// TIA Portal V16 export
// export: Created 2021-11-12T13:32:42.386026Z, ExportSetting WithDefaults, DisplayName Totally Integrated Automation Portal, DisplayVersion V16 Update 3, DisplayName TIA Portal Version Control Interface, DisplayVersion V16 Update 2, DisplayName TIA Portal Openness, DisplayVersion V16 Update 3, DisplayName SINAMICS Startdrive Advanced, DisplayVersion V16 Update 5, DisplayName SINAMICS Startdrive G130, G150, S120, S150, SINAMICS MV, S210, DisplayVersion V16 Update 5, DisplayName SINAMICS Startdrive G110M, G120, G120C, G120D, G120P, G115D, DisplayVersion V16 Update 5, DisplayName STEP 7 Professional, DisplayVersion V16 Update 3, DisplayName STEP 7 Safety, DisplayVersion V16, DisplayName WinCC UA Professional, DisplayVersion V16 Update 3
FUNCTION_BLOCK "StationSCH1"   // FB25, LAD
{ S7_Optimized_Access := 'TRUE' }
VERSION : 0.1
// stored: AutoNumber true, IsIECCheckEnabled false, IsRetainMemResEnabled false, MemoryReserve 100, SetENOAutomatically false, UDAEnableTagReadback false
   VAR_INPUT
      IS_Inputs : "UDT_COMM_SCH1_CRS";
   END_VAR
   VAR_OUTPUT
      OS_Outputs : "UDT_COMM_CRS_SCH1";
      OS_Status : "UDT_SCH_Status_specific";
   END_VAR
   VAR_IN_OUT
      XS_Parameter : "UDT_SCH_Parameter";
      XS_HMICommand : "UDT_SCH_Command";
   END_VAR
   VAR
      SF_Alarm1 : "STD_DI_Mon";
      SF_Alarm2 : "STD_DI_Mon";
      SF_Alarm3 : "STD_DI_Mon";
      SF_Alarm4 : "STD_DI_Mon";
      SF_Alarm5 : "STD_DI_Mon";
      SF_Alarm6 : "STD_DI_Mon";
      SF_Alarm7 : "STD_DI_Mon";
      SF_Alarm8 : "STD_DI_Mon";
      SF_Alarm9 : "STD_DI_Mon";
      SF_QW180 { S7_SetPoint := 'True'} : "STD_CH_AO";
      SF_QW182 { S7_SetPoint := 'True'} : "STD_CH_AO";
      SF_QW184 { S7_SetPoint := 'True'} : "STD_CH_AO";
      SF_QW186 { S7_SetPoint := 'True'} : "STD_CH_AO";
      Edge { S7_SetPoint := 'True'} : Array[0..31] of Bool;   // Edge evalution
      ST_Die3Rdy : TON_TIME;
      ST_Die456Rdy : TON_TIME;
      ST_StartPulse { S7_SetPoint := 'True'} : TP_TIME;
   END_VAR
   VAR RETAIN
      SDI_PartID : DInt;
      SI_PartType : Int;
   END_VAR
   VAR
      SF_Alarm10 { S7_SetPoint := 'True'} : "STD_DI_Mon";
   END_VAR
   VAR_TEMP
      TB1PwrOk : Bool;
      TB1_ReqOnePart : Bool;   // Request to eject one part
      TB1_ReqAllParts : Bool;   // Request to eject all parts in row
      TI_BufferFreePos : Int;   // Number of free position in buffer
      TI_Index1 : Int;   // Index
      TI_Index2 : Int;   // Index
      TS_Parameter : "UDT_SCH_Parameter";
      TS_HMICommand : "UDT_SCH_Command";
      TR_TempUpperLim : Real;   // Upper limit of tool temperature
      TR_TempLowerLim : Real;   // Lower limit of tool temperature
      TDI_BrakeTestTime : DInt;   // Remaining time to brake test - Press [min]
   END_VAR
   VAR CONSTANT
      CT_DieRdy : Time := T#5m;
      CT_StartPulse : Time := T#1s;
      CR_BrakeTestWrn : Real := 10.0;   // [min]
   END_VAR
   VAR_TEMP   // added for the SCL form of the ladder/FBD networks
      _w1 : Bool;
      _w2 : Bool;
      _w3 : Bool;
      _w4 : Bool;
      _w5 : Bool;
      _w6 : Bool;
      _w7 : Bool;
      _w8 : Bool;
      _w9 : Bool;
      _w10 : Bool;
      _w11 : Bool;
      _w12 : Bool;
      _w13 : Bool;
      _w14 : Bool;
      _w15 : Bool;
   END_VAR
BEGIN

REGION Network 1: Clear temporary variables
END_REGION

REGION Network 2: Copy In/Out variables to temporary variables
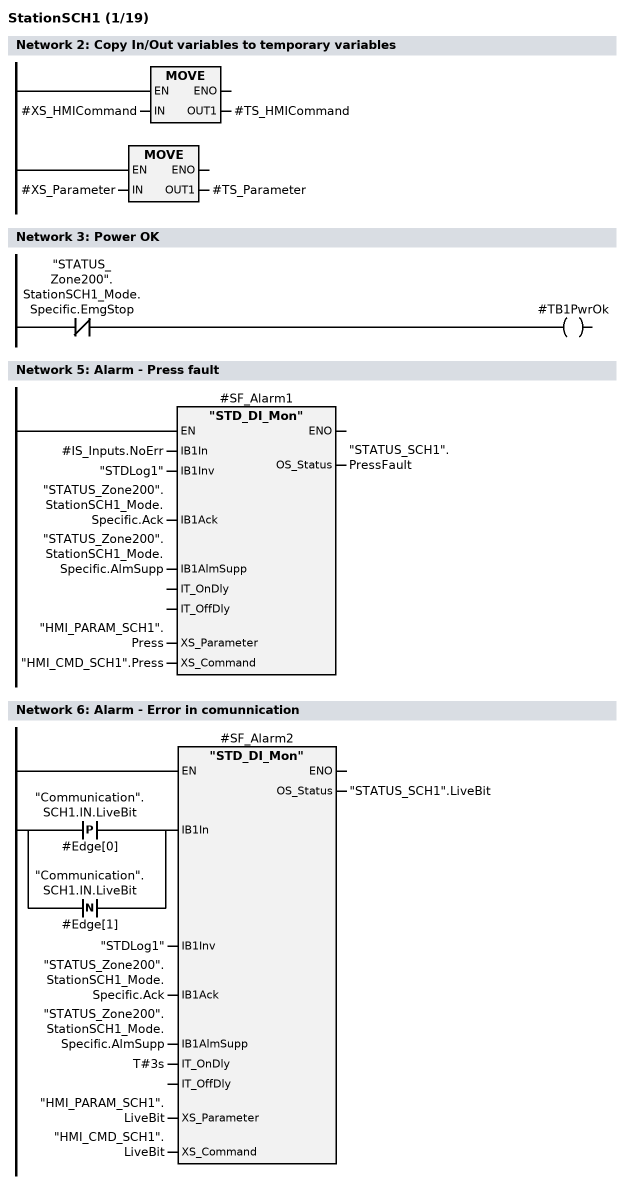
   RUNG wire#powerrail
      Move(in := #XS_HMICommand, out1 => #TS_HMICommand)
   END_RUNG
   RUNG wire#powerrail
      Move(in := #XS_Parameter, out1 => #TS_Parameter)
   END_RUNG
   // the same network as SCL:
   #TS_HMICommand := #XS_HMICommand;
   #TS_Parameter := #XS_Parameter;
END_REGION

REGION Network 3: Power OK
   RUNG wire#powerrail
      I_Contact( "STATUS_Zone200".StationSCH1_Mode.Specific.EmgStop )
      Coil( #TB1PwrOk )
   END_RUNG
   // the same network as SCL:
   #TB1PwrOk := NOT "STATUS_Zone200".StationSCH1_Mode.Specific.EmgStop;
END_REGION

REGION Network 4: *************** Alarms ***************
END_REGION

REGION Network 5: Alarm - Press fault
   RUNG wire#powerrail
      #SF_Alarm1(IB1In := #IS_Inputs.NoErr, IB1Inv := "STDLog1", IB1Ack := "STATUS_Zone200".StationSCH1_Mode.Specific.Ack, IB1AlmSupp := "STATUS_Zone200".StationSCH1_Mode.Specific.AlmSupp, IT_OnDly :=, IT_OffDly :=, XS_Parameter := "HMI_PARAM_SCH1".Press, XS_Command := "HMI_CMD_SCH1".Press, OS_Status => "STATUS_SCH1".PressFault)
   END_RUNG
   // the same network as SCL:
   #SF_Alarm1(IB1In := #IS_Inputs.NoErr,   // "STD_DI_Mon"
              IB1Inv := "STDLog1",
              IB1Ack := "STATUS_Zone200".StationSCH1_Mode.Specific.Ack,
              IB1AlmSupp := "STATUS_Zone200".StationSCH1_Mode.Specific.AlmSupp,
              XS_Parameter := "HMI_PARAM_SCH1".Press,
              XS_Command := "HMI_CMD_SCH1".Press,
              OS_Status => "STATUS_SCH1".PressFault);
END_REGION

REGION Network 6: Alarm - Error in comunnication
   RUNG wire#powerrail
      #SF_Alarm2(IB1In := wire#w1, IB1Inv := "STDLog1", IB1Ack := "STATUS_Zone200".StationSCH1_Mode.Specific.Ack, IB1AlmSupp := "STATUS_Zone200".StationSCH1_Mode.Specific.AlmSupp, IT_OnDly := T#3s, IT_OffDly :=, XS_Parameter := "HMI_PARAM_SCH1".LiveBit, XS_Command := "HMI_CMD_SCH1".LiveBit, OS_Status => "STATUS_SCH1".LiveBit)
   END_RUNG
   RUNG wire#powerrail
      P_Contact(operand := "Communication".SCH1.IN.LiveBit, bit := #Edge[0])
   END_RUNG wire#w1
   RUNG wire#powerrail
      N_Contact(operand := "Communication".SCH1.IN.LiveBit, bit := #Edge[1])
   END_RUNG wire#w1
   // the same network as SCL:
   #_w1 := "Communication".SCH1.IN.LiveBit AND NOT #Edge[0];   // rising edge of "Communication".SCH1.IN.LiveBit
   #Edge[0] := "Communication".SCH1.IN.LiveBit;
   #_w2 := NOT "Communication".SCH1.IN.LiveBit AND #Edge[1];   // falling edge of "Communication".SCH1.IN.LiveBit
   #Edge[1] := "Communication".SCH1.IN.LiveBit;
   #SF_Alarm2(IB1In := #_w1 OR #_w2,   // "STD_DI_Mon"
              IB1Inv := "STDLog1",
              IB1Ack := "STATUS_Zone200".StationSCH1_Mode.Specific.Ack,
              IB1AlmSupp := "STATUS_Zone200".StationSCH1_Mode.Specific.AlmSupp,
              IT_OnDly := T#3s,
              XS_Parameter := "HMI_PARAM_SCH1".LiveBit,
              XS_Command := "HMI_CMD_SCH1".LiveBit,
              OS_Status => "STATUS_SCH1".LiveBit);
END_REGION

REGION Network 7: Alarm - Tool heating 1 up - temperature is out of tolerance
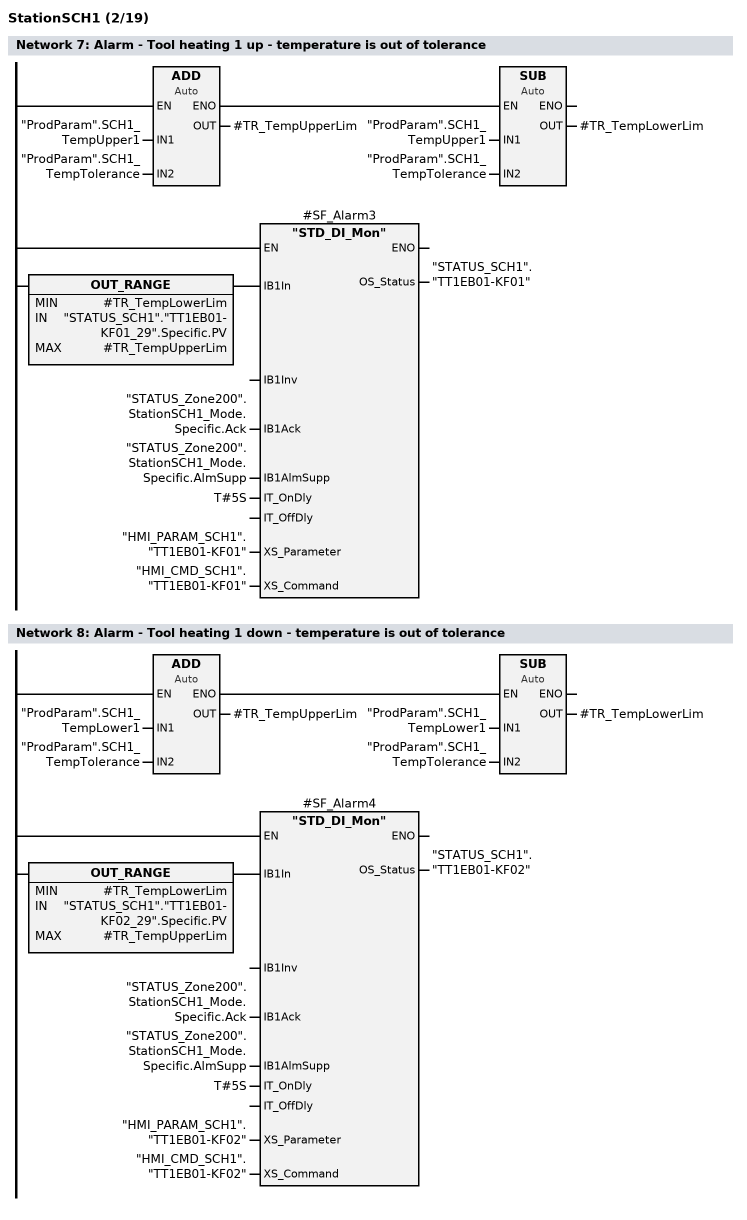
   #TR_TempUpperLim := "ProdParam".SCH1_TempUpper1 + "ProdParam".SCH1_TempTolerance;
   #TR_TempLowerLim := "ProdParam".SCH1_TempUpper1 - "ProdParam".SCH1_TempTolerance;
   #SF_Alarm3(IB1In := ("STATUS_SCH1"."TT1EB01-KF01_29".Specific.PV < #TR_TempLowerLim) OR ("STATUS_SCH1"."TT1EB01-KF01_29".Specific.PV > #TR_TempUpperLim),   // "STD_DI_Mon"
              IB1Ack := "STATUS_Zone200".StationSCH1_Mode.Specific.Ack,
              IB1AlmSupp := "STATUS_Zone200".StationSCH1_Mode.Specific.AlmSupp,
              IT_OnDly := T#5S,
              XS_Parameter := "HMI_PARAM_SCH1"."TT1EB01-KF01",
              XS_Command := "HMI_CMD_SCH1"."TT1EB01-KF01",
              OS_Status => "STATUS_SCH1"."TT1EB01-KF01");
END_REGION

REGION Network 8: Alarm - Tool heating 1 down - temperature is out of tolerance
   #TR_TempUpperLim := "ProdParam".SCH1_TempLower1 + "ProdParam".SCH1_TempTolerance;
   #TR_TempLowerLim := "ProdParam".SCH1_TempLower1 - "ProdParam".SCH1_TempTolerance;
   #SF_Alarm4(IB1In := ("STATUS_SCH1"."TT1EB01-KF02_29".Specific.PV < #TR_TempLowerLim) OR ("STATUS_SCH1"."TT1EB01-KF02_29".Specific.PV > #TR_TempUpperLim),   // "STD_DI_Mon"
              IB1Ack := "STATUS_Zone200".StationSCH1_Mode.Specific.Ack,
              IB1AlmSupp := "STATUS_Zone200".StationSCH1_Mode.Specific.AlmSupp,
              IT_OnDly := T#5S,
              XS_Parameter := "HMI_PARAM_SCH1"."TT1EB01-KF02",
              XS_Command := "HMI_CMD_SCH1"."TT1EB01-KF02",
              OS_Status => "STATUS_SCH1"."TT1EB01-KF02");
END_REGION

REGION Network 9: Alarm - Tool heating 2 up - temperature is out of tolerance
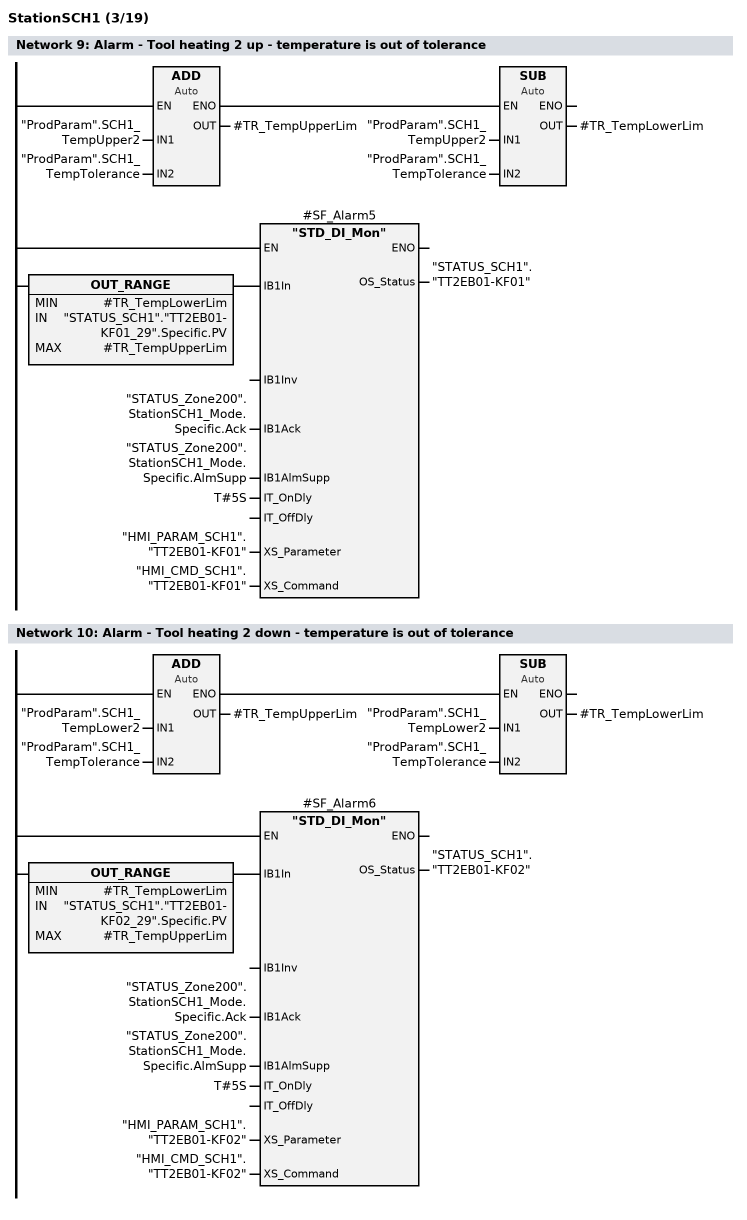
   #TR_TempUpperLim := "ProdParam".SCH1_TempUpper2 + "ProdParam".SCH1_TempTolerance;
   #TR_TempLowerLim := "ProdParam".SCH1_TempUpper2 - "ProdParam".SCH1_TempTolerance;
   #SF_Alarm5(IB1In := ("STATUS_SCH1"."TT2EB01-KF01_29".Specific.PV < #TR_TempLowerLim) OR ("STATUS_SCH1"."TT2EB01-KF01_29".Specific.PV > #TR_TempUpperLim),   // "STD_DI_Mon"
              IB1Ack := "STATUS_Zone200".StationSCH1_Mode.Specific.Ack,
              IB1AlmSupp := "STATUS_Zone200".StationSCH1_Mode.Specific.AlmSupp,
              IT_OnDly := T#5S,
              XS_Parameter := "HMI_PARAM_SCH1"."TT2EB01-KF01",
              XS_Command := "HMI_CMD_SCH1"."TT2EB01-KF01",
              OS_Status => "STATUS_SCH1"."TT2EB01-KF01");
END_REGION

REGION Network 10: Alarm - Tool heating 2 down - temperature is out of tolerance
   #TR_TempUpperLim := "ProdParam".SCH1_TempLower2 + "ProdParam".SCH1_TempTolerance;
   #TR_TempLowerLim := "ProdParam".SCH1_TempLower2 - "ProdParam".SCH1_TempTolerance;
   #SF_Alarm6(IB1In := ("STATUS_SCH1"."TT2EB01-KF02_29".Specific.PV < #TR_TempLowerLim) OR ("STATUS_SCH1"."TT2EB01-KF02_29".Specific.PV > #TR_TempUpperLim),   // "STD_DI_Mon"
              IB1Ack := "STATUS_Zone200".StationSCH1_Mode.Specific.Ack,
              IB1AlmSupp := "STATUS_Zone200".StationSCH1_Mode.Specific.AlmSupp,
              IT_OnDly := T#5S,
              XS_Parameter := "HMI_PARAM_SCH1"."TT2EB01-KF02",
              XS_Command := "HMI_CMD_SCH1"."TT2EB01-KF02",
              OS_Status => "STATUS_SCH1"."TT2EB01-KF02");
END_REGION

REGION Network 11: Alarm - Tool heating 1 - pump not running
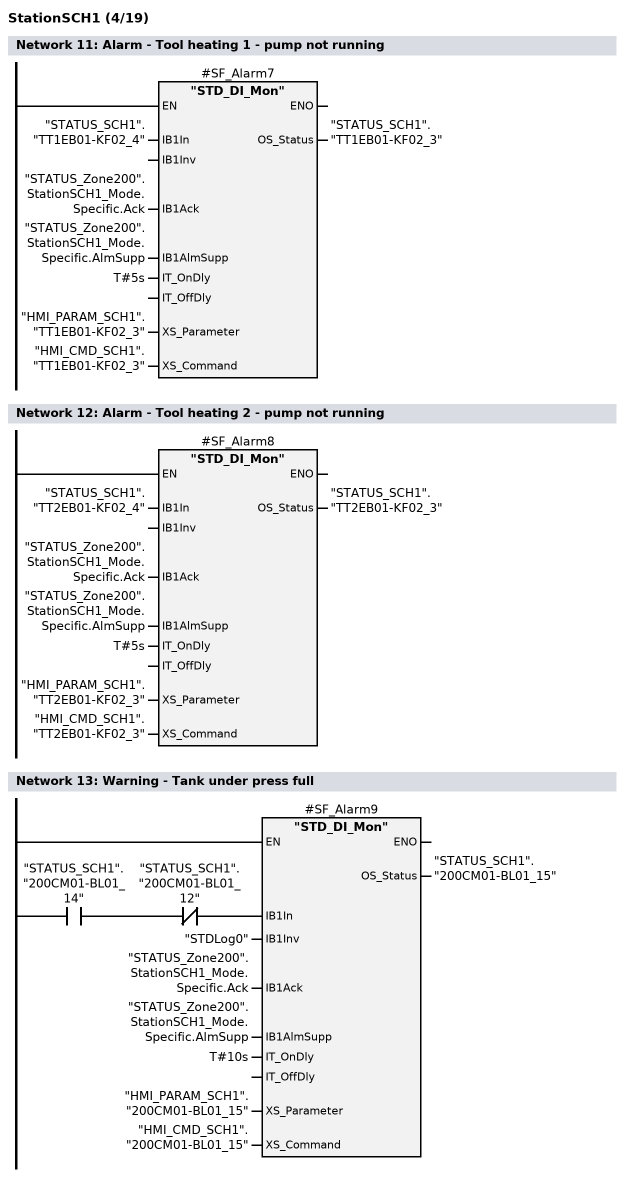
   RUNG wire#powerrail
      #SF_Alarm7(IB1In := "STATUS_SCH1"."TT1EB01-KF02_4", IB1Inv :=, IB1Ack := "STATUS_Zone200".StationSCH1_Mode.Specific.Ack, IB1AlmSupp := "STATUS_Zone200".StationSCH1_Mode.Specific.AlmSupp, IT_OnDly := T#5s, IT_OffDly :=, XS_Parameter := "HMI_PARAM_SCH1"."TT1EB01-KF02_3", XS_Command := "HMI_CMD_SCH1"."TT1EB01-KF02_3", OS_Status => "STATUS_SCH1"."TT1EB01-KF02_3")
   END_RUNG
   // the same network as SCL:
   #SF_Alarm7(IB1In := "STATUS_SCH1"."TT1EB01-KF02_4",   // "STD_DI_Mon"
              IB1Ack := "STATUS_Zone200".StationSCH1_Mode.Specific.Ack,
              IB1AlmSupp := "STATUS_Zone200".StationSCH1_Mode.Specific.AlmSupp,
              IT_OnDly := T#5s,
              XS_Parameter := "HMI_PARAM_SCH1"."TT1EB01-KF02_3",
              XS_Command := "HMI_CMD_SCH1"."TT1EB01-KF02_3",
              OS_Status => "STATUS_SCH1"."TT1EB01-KF02_3");
END_REGION

REGION Network 12: Alarm - Tool heating 2 - pump not running
   RUNG wire#powerrail
      #SF_Alarm8(IB1In := "STATUS_SCH1"."TT2EB01-KF02_4", IB1Inv :=, IB1Ack := "STATUS_Zone200".StationSCH1_Mode.Specific.Ack, IB1AlmSupp := "STATUS_Zone200".StationSCH1_Mode.Specific.AlmSupp, IT_OnDly := T#5s, IT_OffDly :=, XS_Parameter := "HMI_PARAM_SCH1"."TT2EB01-KF02_3", XS_Command := "HMI_CMD_SCH1"."TT2EB01-KF02_3", OS_Status => "STATUS_SCH1"."TT2EB01-KF02_3")
   END_RUNG
   // the same network as SCL:
   #SF_Alarm8(IB1In := "STATUS_SCH1"."TT2EB01-KF02_4",   // "STD_DI_Mon"
              IB1Ack := "STATUS_Zone200".StationSCH1_Mode.Specific.Ack,
              IB1AlmSupp := "STATUS_Zone200".StationSCH1_Mode.Specific.AlmSupp,
              IT_OnDly := T#5s,
              XS_Parameter := "HMI_PARAM_SCH1"."TT2EB01-KF02_3",
              XS_Command := "HMI_CMD_SCH1"."TT2EB01-KF02_3",
              OS_Status => "STATUS_SCH1"."TT2EB01-KF02_3");
END_REGION

REGION Network 13: Warning - Tank under press full
   RUNG wire#powerrail
      #SF_Alarm9(IB1In := wire#w1, IB1Inv := "STDLog0", IB1Ack := "STATUS_Zone200".StationSCH1_Mode.Specific.Ack, IB1AlmSupp := "STATUS_Zone200".StationSCH1_Mode.Specific.AlmSupp, IT_OnDly := T#10s, IT_OffDly :=, XS_Parameter := "HMI_PARAM_SCH1"."200CM01-BL01_15", XS_Command := "HMI_CMD_SCH1"."200CM01-BL01_15", OS_Status => "STATUS_SCH1"."200CM01-BL01_15")
   END_RUNG
   RUNG wire#powerrail
      Contact( "STATUS_SCH1"."200CM01-BL01_14" )
      I_Contact( "STATUS_SCH1"."200CM01-BL01_12" )
   END_RUNG wire#w1
   // the same network as SCL:
   #SF_Alarm9(IB1In := "STATUS_SCH1"."200CM01-BL01_14" AND NOT "STATUS_SCH1"."200CM01-BL01_12",   // "STD_DI_Mon"
              IB1Inv := "STDLog0",
              IB1Ack := "STATUS_Zone200".StationSCH1_Mode.Specific.Ack,
              IB1AlmSupp := "STATUS_Zone200".StationSCH1_Mode.Specific.AlmSupp,
              IT_OnDly := T#10s,
              XS_Parameter := "HMI_PARAM_SCH1"."200CM01-BL01_15",
              XS_Command := "HMI_CMD_SCH1"."200CM01-BL01_15",
              OS_Status => "STATUS_SCH1"."200CM01-BL01_15");
END_REGION

REGION Network 14: Warning - Brake test required
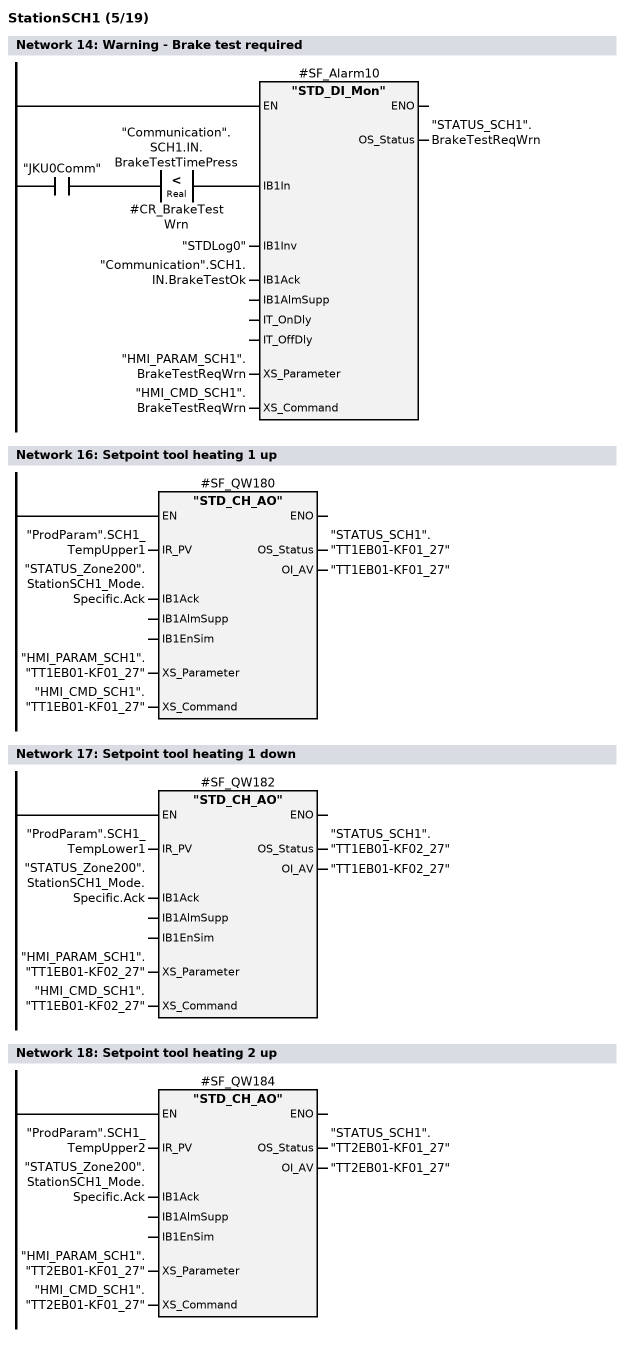
   RUNG wire#powerrail
      #SF_Alarm10(IB1In := wire#w1, IB1Inv := "STDLog0", IB1Ack := "Communication".SCH1.IN.BrakeTestOk, IB1AlmSupp :=, IT_OnDly :=, IT_OffDly :=, XS_Parameter := "HMI_PARAM_SCH1".BrakeTestReqWrn, XS_Command := "HMI_CMD_SCH1".BrakeTestReqWrn, OS_Status => "STATUS_SCH1".BrakeTestReqWrn)
   END_RUNG
   RUNG wire#powerrail
      Contact( "JKU0Comm" )
      { S7_Templates := "SrcType := Real" } LT_Contact(in1 := "Communication".SCH1.IN.BrakeTestTimePress, in2 := #CR_BrakeTestWrn)
   END_RUNG wire#w1
   // the same network as SCL:
   #SF_Alarm10(IB1In := "JKU0Comm" AND ("Communication".SCH1.IN.BrakeTestTimePress < #CR_BrakeTestWrn),   // "STD_DI_Mon"
               IB1Inv := "STDLog0",
               IB1Ack := "Communication".SCH1.IN.BrakeTestOk,
               XS_Parameter := "HMI_PARAM_SCH1".BrakeTestReqWrn,
               XS_Command := "HMI_CMD_SCH1".BrakeTestReqWrn,
               OS_Status => "STATUS_SCH1".BrakeTestReqWrn);
END_REGION

REGION Network 15: *************** Tool temperature setpoints ***************
END_REGION

REGION Network 16: Setpoint tool heating 1 up
   RUNG wire#powerrail
      #SF_QW180(IR_PV := "ProdParam".SCH1_TempUpper1, IB1Ack := "STATUS_Zone200".StationSCH1_Mode.Specific.Ack, IB1AlmSupp :=, IB1EnSim :=, XS_Parameter := "HMI_PARAM_SCH1"."TT1EB01-KF01_27", XS_Command := "HMI_CMD_SCH1"."TT1EB01-KF01_27", OS_Status => "STATUS_SCH1"."TT1EB01-KF01_27", OI_AV => "TT1EB01-KF01_27")
   END_RUNG
   // the same network as SCL:
   #SF_QW180(IR_PV := "ProdParam".SCH1_TempUpper1,   // "STD_CH_AO"
             IB1Ack := "STATUS_Zone200".StationSCH1_Mode.Specific.Ack,
             XS_Parameter := "HMI_PARAM_SCH1"."TT1EB01-KF01_27",
             XS_Command := "HMI_CMD_SCH1"."TT1EB01-KF01_27",
             OS_Status => "STATUS_SCH1"."TT1EB01-KF01_27",
             OI_AV => "TT1EB01-KF01_27");
END_REGION

REGION Network 17: Setpoint tool heating 1 down
   RUNG wire#powerrail
      #SF_QW182(IR_PV := "ProdParam".SCH1_TempLower1, IB1Ack := "STATUS_Zone200".StationSCH1_Mode.Specific.Ack, IB1AlmSupp :=, IB1EnSim :=, XS_Parameter := "HMI_PARAM_SCH1"."TT1EB01-KF02_27", XS_Command := "HMI_CMD_SCH1"."TT1EB01-KF02_27", OS_Status => "STATUS_SCH1"."TT1EB01-KF02_27", OI_AV => "TT1EB01-KF02_27")
   END_RUNG
   // the same network as SCL:
   #SF_QW182(IR_PV := "ProdParam".SCH1_TempLower1,   // "STD_CH_AO"
             IB1Ack := "STATUS_Zone200".StationSCH1_Mode.Specific.Ack,
             XS_Parameter := "HMI_PARAM_SCH1"."TT1EB01-KF02_27",
             XS_Command := "HMI_CMD_SCH1"."TT1EB01-KF02_27",
             OS_Status => "STATUS_SCH1"."TT1EB01-KF02_27",
             OI_AV => "TT1EB01-KF02_27");
END_REGION

REGION Network 18: Setpoint tool heating 2 up
   RUNG wire#powerrail
      #SF_QW184(IR_PV := "ProdParam".SCH1_TempUpper2, IB1Ack := "STATUS_Zone200".StationSCH1_Mode.Specific.Ack, IB1AlmSupp :=, IB1EnSim :=, XS_Parameter := "HMI_PARAM_SCH1"."TT2EB01-KF01_27", XS_Command := "HMI_CMD_SCH1"."TT2EB01-KF01_27", OS_Status => "STATUS_SCH1"."TT2EB01-KF01_27", OI_AV => "TT2EB01-KF01_27")
   END_RUNG
   // the same network as SCL:
   #SF_QW184(IR_PV := "ProdParam".SCH1_TempUpper2,   // "STD_CH_AO"
             IB1Ack := "STATUS_Zone200".StationSCH1_Mode.Specific.Ack,
             XS_Parameter := "HMI_PARAM_SCH1"."TT2EB01-KF01_27",
             XS_Command := "HMI_CMD_SCH1"."TT2EB01-KF01_27",
             OS_Status => "STATUS_SCH1"."TT2EB01-KF01_27",
             OI_AV => "TT2EB01-KF01_27");
END_REGION

REGION Network 19: Setpoint tool heating 2 down
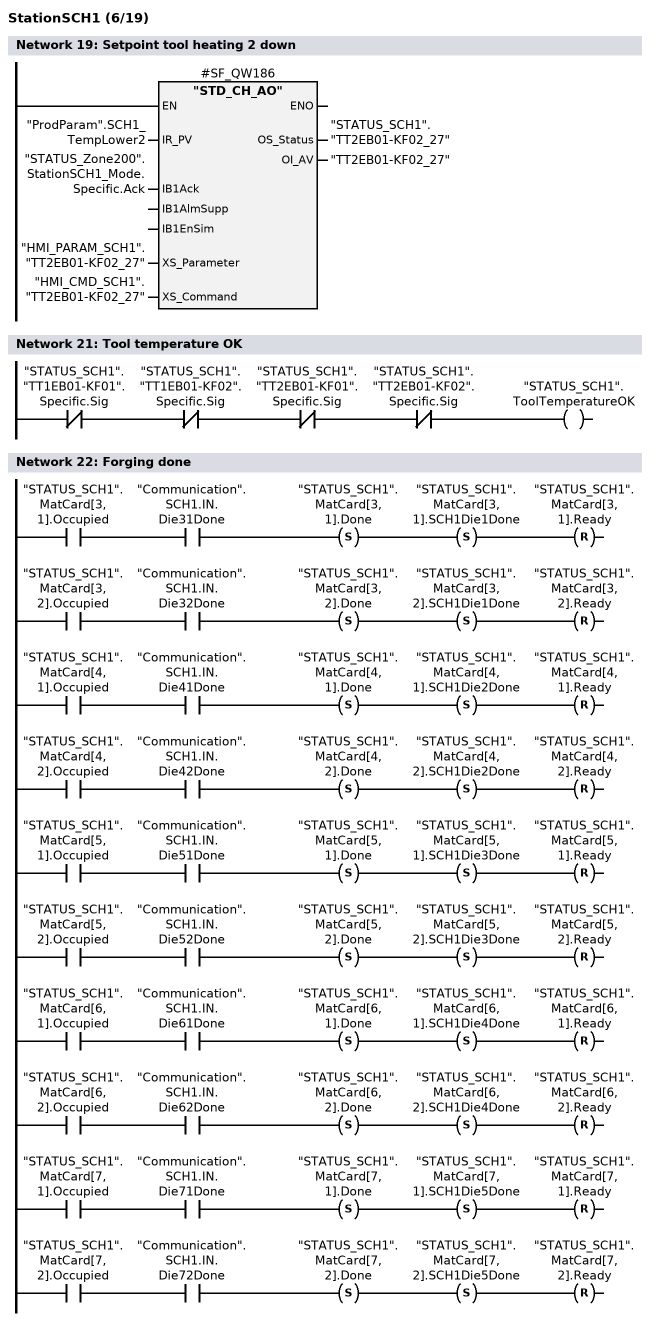
   RUNG wire#powerrail
      #SF_QW186(IR_PV := "ProdParam".SCH1_TempLower2, IB1Ack := "STATUS_Zone200".StationSCH1_Mode.Specific.Ack, IB1AlmSupp :=, IB1EnSim :=, XS_Parameter := "HMI_PARAM_SCH1"."TT2EB01-KF02_27", XS_Command := "HMI_CMD_SCH1"."TT2EB01-KF02_27", OS_Status => "STATUS_SCH1"."TT2EB01-KF02_27", OI_AV => "TT2EB01-KF02_27")
   END_RUNG
   // the same network as SCL:
   #SF_QW186(IR_PV := "ProdParam".SCH1_TempLower2,   // "STD_CH_AO"
             IB1Ack := "STATUS_Zone200".StationSCH1_Mode.Specific.Ack,
             XS_Parameter := "HMI_PARAM_SCH1"."TT2EB01-KF02_27",
             XS_Command := "HMI_CMD_SCH1"."TT2EB01-KF02_27",
             OS_Status => "STATUS_SCH1"."TT2EB01-KF02_27",
             OI_AV => "TT2EB01-KF02_27");
END_REGION

REGION Network 20: *************** States ***************
END_REGION

REGION Network 21: Tool temperature OK
   RUNG wire#powerrail
      I_Contact( "STATUS_SCH1"."TT1EB01-KF01".Specific.Sig )
      I_Contact( "STATUS_SCH1"."TT1EB01-KF02".Specific.Sig )
      I_Contact( "STATUS_SCH1"."TT2EB01-KF01".Specific.Sig )
      I_Contact( "STATUS_SCH1"."TT2EB01-KF02".Specific.Sig )
      Coil( "STATUS_SCH1".ToolTemperatureOK )
   END_RUNG
   // the same network as SCL:
   "STATUS_SCH1".ToolTemperatureOK := NOT "STATUS_SCH1"."TT1EB01-KF01".Specific.Sig AND NOT "STATUS_SCH1"."TT1EB01-KF02".Specific.Sig AND NOT "STATUS_SCH1"."TT2EB01-KF01".Specific.Sig AND NOT "STATUS_SCH1"."TT2EB01-KF02".Specific.Sig;
END_REGION

REGION Network 22: Forging done
   RUNG wire#powerrail
      Contact( "STATUS_SCH1".MatCard[3, 1].Occupied )
      Contact( "Communication".SCH1.IN.Die31Done )
      S_Coil( "STATUS_SCH1".MatCard[3, 1].Done )
      S_Coil( "STATUS_SCH1".MatCard[3, 1].SCH1Die1Done )
      R_Coil( "STATUS_SCH1".MatCard[3, 1].Ready )
   END_RUNG
   RUNG wire#powerrail
      Contact( "STATUS_SCH1".MatCard[3, 2].Occupied )
      Contact( "Communication".SCH1.IN.Die32Done )
      S_Coil( "STATUS_SCH1".MatCard[3, 2].Done )
      S_Coil( "STATUS_SCH1".MatCard[3, 2].SCH1Die1Done )
      R_Coil( "STATUS_SCH1".MatCard[3, 2].Ready )
   END_RUNG
   RUNG wire#powerrail
      Contact( "STATUS_SCH1".MatCard[4, 1].Occupied )
      Contact( "Communication".SCH1.IN.Die41Done )
      S_Coil( "STATUS_SCH1".MatCard[4, 1].Done )
      S_Coil( "STATUS_SCH1".MatCard[4, 1].SCH1Die2Done )
      R_Coil( "STATUS_SCH1".MatCard[4, 1].Ready )
   END_RUNG
   RUNG wire#powerrail
      Contact( "STATUS_SCH1".MatCard[4, 2].Occupied )
      Contact( "Communication".SCH1.IN.Die42Done )
      S_Coil( "STATUS_SCH1".MatCard[4, 2].Done )
      S_Coil( "STATUS_SCH1".MatCard[4, 2].SCH1Die2Done )
      R_Coil( "STATUS_SCH1".MatCard[4, 2].Ready )
   END_RUNG
   RUNG wire#powerrail
      Contact( "STATUS_SCH1".MatCard[5, 1].Occupied )
      Contact( "Communication".SCH1.IN.Die51Done )
      S_Coil( "STATUS_SCH1".MatCard[5, 1].Done )
      S_Coil( "STATUS_SCH1".MatCard[5, 1].SCH1Die3Done )
      R_Coil( "STATUS_SCH1".MatCard[5, 1].Ready )
   END_RUNG
   RUNG wire#powerrail
      Contact( "STATUS_SCH1".MatCard[5, 2].Occupied )
      Contact( "Communication".SCH1.IN.Die52Done )
      S_Coil( "STATUS_SCH1".MatCard[5, 2].Done )
      S_Coil( "STATUS_SCH1".MatCard[5, 2].SCH1Die3Done )
      R_Coil( "STATUS_SCH1".MatCard[5, 2].Ready )
   END_RUNG
   RUNG wire#powerrail
      Contact( "STATUS_SCH1".MatCard[6, 1].Occupied )
      Contact( "Communication".SCH1.IN.Die61Done )
      S_Coil( "STATUS_SCH1".MatCard[6, 1].Done )
      S_Coil( "STATUS_SCH1".MatCard[6, 1].SCH1Die4Done )
      R_Coil( "STATUS_SCH1".MatCard[6, 1].Ready )
   END_RUNG
   RUNG wire#powerrail
      Contact( "STATUS_SCH1".MatCard[6, 2].Occupied )
      Contact( "Communication".SCH1.IN.Die62Done )
      S_Coil( "STATUS_SCH1".MatCard[6, 2].Done )
      S_Coil( "STATUS_SCH1".MatCard[6, 2].SCH1Die4Done )
      R_Coil( "STATUS_SCH1".MatCard[6, 2].Ready )
   END_RUNG
   RUNG wire#powerrail
      Contact( "STATUS_SCH1".MatCard[7, 1].Occupied )
      Contact( "Communication".SCH1.IN.Die71Done )
      S_Coil( "STATUS_SCH1".MatCard[7, 1].Done )
      S_Coil( "STATUS_SCH1".MatCard[7, 1].SCH1Die5Done )
      R_Coil( "STATUS_SCH1".MatCard[7, 1].Ready )
   END_RUNG
   RUNG wire#powerrail
      Contact( "STATUS_SCH1".MatCard[7, 2].Occupied )
      Contact( "Communication".SCH1.IN.Die72Done )
      S_Coil( "STATUS_SCH1".MatCard[7, 2].Done )
      S_Coil( "STATUS_SCH1".MatCard[7, 2].SCH1Die5Done )
      R_Coil( "STATUS_SCH1".MatCard[7, 2].Ready )
   END_RUNG
   // the same network as SCL:
   #_w1 := "STATUS_SCH1".MatCard[3, 1].Occupied AND "Communication".SCH1.IN.Die31Done;
   IF #_w1 THEN
       "STATUS_SCH1".MatCard[3, 1].Done := TRUE;
       "STATUS_SCH1".MatCard[3, 1].SCH1Die1Done := TRUE;
       "STATUS_SCH1".MatCard[3, 1].Ready := FALSE;
   END_IF;
   #_w2 := "STATUS_SCH1".MatCard[3, 2].Occupied AND "Communication".SCH1.IN.Die32Done;
   IF #_w2 THEN
       "STATUS_SCH1".MatCard[3, 2].Done := TRUE;
       "STATUS_SCH1".MatCard[3, 2].SCH1Die1Done := TRUE;
       "STATUS_SCH1".MatCard[3, 2].Ready := FALSE;
   END_IF;
   #_w3 := "STATUS_SCH1".MatCard[4, 1].Occupied AND "Communication".SCH1.IN.Die41Done;
   IF #_w3 THEN
       "STATUS_SCH1".MatCard[4, 1].Done := TRUE;
       "STATUS_SCH1".MatCard[4, 1].SCH1Die2Done := TRUE;
       "STATUS_SCH1".MatCard[4, 1].Ready := FALSE;
   END_IF;
   #_w4 := "STATUS_SCH1".MatCard[4, 2].Occupied AND "Communication".SCH1.IN.Die42Done;
   IF #_w4 THEN
       "STATUS_SCH1".MatCard[4, 2].Done := TRUE;
       "STATUS_SCH1".MatCard[4, 2].SCH1Die2Done := TRUE;
       "STATUS_SCH1".MatCard[4, 2].Ready := FALSE;
   END_IF;
   #_w5 := "STATUS_SCH1".MatCard[5, 1].Occupied AND "Communication".SCH1.IN.Die51Done;
   IF #_w5 THEN
       "STATUS_SCH1".MatCard[5, 1].Done := TRUE;
       "STATUS_SCH1".MatCard[5, 1].SCH1Die3Done := TRUE;
       "STATUS_SCH1".MatCard[5, 1].Ready := FALSE;
   END_IF;
   #_w6 := "STATUS_SCH1".MatCard[5, 2].Occupied AND "Communication".SCH1.IN.Die52Done;
   IF #_w6 THEN
       "STATUS_SCH1".MatCard[5, 2].Done := TRUE;
       "STATUS_SCH1".MatCard[5, 2].SCH1Die3Done := TRUE;
       "STATUS_SCH1".MatCard[5, 2].Ready := FALSE;
   END_IF;
   #_w7 := "STATUS_SCH1".MatCard[6, 1].Occupied AND "Communication".SCH1.IN.Die61Done;
   IF #_w7 THEN
       "STATUS_SCH1".MatCard[6, 1].Done := TRUE;
       "STATUS_SCH1".MatCard[6, 1].SCH1Die4Done := TRUE;
       "STATUS_SCH1".MatCard[6, 1].Ready := FALSE;
   END_IF;
   #_w8 := "STATUS_SCH1".MatCard[6, 2].Occupied AND "Communication".SCH1.IN.Die62Done;
   IF #_w8 THEN
       "STATUS_SCH1".MatCard[6, 2].Done := TRUE;
       "STATUS_SCH1".MatCard[6, 2].SCH1Die4Done := TRUE;
       "STATUS_SCH1".MatCard[6, 2].Ready := FALSE;
   END_IF;
   #_w9 := "STATUS_SCH1".MatCard[7, 1].Occupied AND "Communication".SCH1.IN.Die71Done;
   IF #_w9 THEN
       "STATUS_SCH1".MatCard[7, 1].Done := TRUE;
       "STATUS_SCH1".MatCard[7, 1].SCH1Die5Done := TRUE;
       "STATUS_SCH1".MatCard[7, 1].Ready := FALSE;
   END_IF;
   #_w10 := "STATUS_SCH1".MatCard[7, 2].Occupied AND "Communication".SCH1.IN.Die72Done;
   IF #_w10 THEN
       "STATUS_SCH1".MatCard[7, 2].Done := TRUE;
       "STATUS_SCH1".MatCard[7, 2].SCH1Die5Done := TRUE;
       "STATUS_SCH1".MatCard[7, 2].Ready := FALSE;
   END_IF;
END_REGION

REGION Network 23 (SCL): Tech. time evaluation
   IF "STDEdge_1s" THEN
       FOR #TI_Index1 := 3 TO 7 DO
           FOR #TI_Index2 := 1 TO 2 DO
               IF "STATUS_SCH1".MatCard[#TI_Index1, #TI_Index2].Occupied THEN
                   "MTS_UpdateTimeInPress"(IB1Clock_1s := "STDEdge_1s",
                                           XS_Position := "STATUS_SCH1".MatCard[#TI_Index1, #TI_Index2]);
               END_IF;
           END_FOR;
       END_FOR;
   END_IF;
END_REGION

REGION Network 24: Output conveyor part counter
END_REGION

REGION Network 25: Brake test time
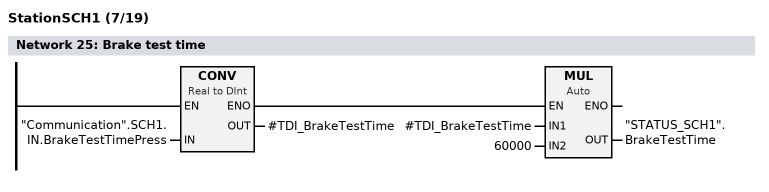
   RUNG wire#powerrail
      { S7_Templates := "[SrcType := Real, DestType := DInt]"; S7_GenerateENO := "TRUE" } Convert(in := "Communication".SCH1.IN.BrakeTestTimePress, out => #TDI_BrakeTestTime)
      { S7_GenerateENO := "TRUE" } Mul(in1 := #TDI_BrakeTestTime, in2 := 60000, out => "STATUS_SCH1".BrakeTestTime)
   END_RUNG
   // the same network as SCL:
   // ENO of a box is taken as its EN; it also drops when the box reports an error
   #TDI_BrakeTestTime := REAL_TO_DINT("Communication".SCH1.IN.BrakeTestTimePress);
   "STATUS_SCH1".BrakeTestTime := #TDI_BrakeTestTime * 60000;
END_REGION

REGION Network 26: *************** Material flow ***************
END_REGION

REGION Network 27: Clear positions and map - commands
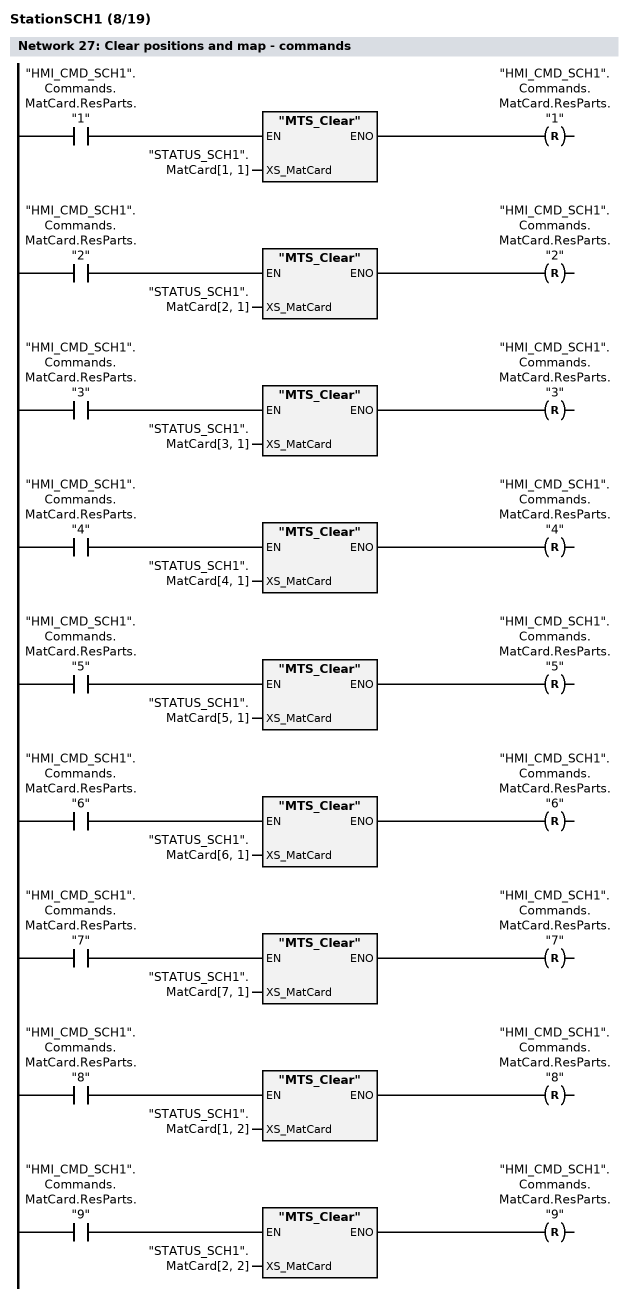
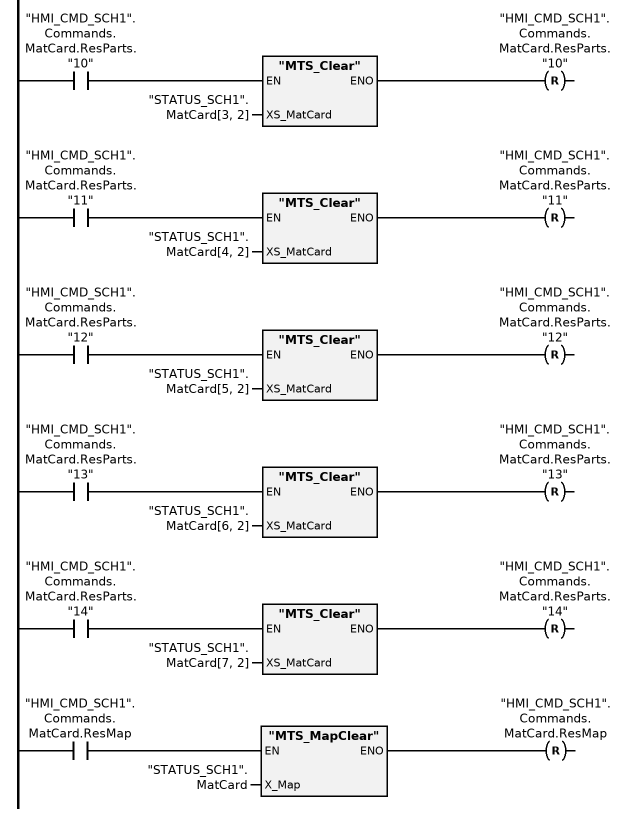
   RUNG wire#powerrail
      Contact( "HMI_CMD_SCH1".Commands.MatCard.ResParts."1" )
      "MTS_Clear"(XS_MatCard := "STATUS_SCH1".MatCard[1, 1])
      R_Coil( "HMI_CMD_SCH1".Commands.MatCard.ResParts."1" )
   END_RUNG
   RUNG wire#powerrail
      Contact( "HMI_CMD_SCH1".Commands.MatCard.ResParts."2" )
      "MTS_Clear"(XS_MatCard := "STATUS_SCH1".MatCard[2, 1])
      R_Coil( "HMI_CMD_SCH1".Commands.MatCard.ResParts."2" )
   END_RUNG
   RUNG wire#powerrail
      Contact( "HMI_CMD_SCH1".Commands.MatCard.ResParts."3" )
      "MTS_Clear"(XS_MatCard := "STATUS_SCH1".MatCard[3, 1])
      R_Coil( "HMI_CMD_SCH1".Commands.MatCard.ResParts."3" )
   END_RUNG
   RUNG wire#powerrail
      Contact( "HMI_CMD_SCH1".Commands.MatCard.ResParts."4" )
      "MTS_Clear"(XS_MatCard := "STATUS_SCH1".MatCard[4, 1])
      R_Coil( "HMI_CMD_SCH1".Commands.MatCard.ResParts."4" )
   END_RUNG
   RUNG wire#powerrail
      Contact( "HMI_CMD_SCH1".Commands.MatCard.ResParts."5" )
      "MTS_Clear"(XS_MatCard := "STATUS_SCH1".MatCard[5, 1])
      R_Coil( "HMI_CMD_SCH1".Commands.MatCard.ResParts."5" )
   END_RUNG
   RUNG wire#powerrail
      Contact( "HMI_CMD_SCH1".Commands.MatCard.ResParts."6" )
      "MTS_Clear"(XS_MatCard := "STATUS_SCH1".MatCard[6, 1])
      R_Coil( "HMI_CMD_SCH1".Commands.MatCard.ResParts."6" )
   END_RUNG
   RUNG wire#powerrail
      Contact( "HMI_CMD_SCH1".Commands.MatCard.ResParts."7" )
      "MTS_Clear"(XS_MatCard := "STATUS_SCH1".MatCard[7, 1])
      R_Coil( "HMI_CMD_SCH1".Commands.MatCard.ResParts."7" )
   END_RUNG
   RUNG wire#powerrail
      Contact( "HMI_CMD_SCH1".Commands.MatCard.ResParts."8" )
      "MTS_Clear"(XS_MatCard := "STATUS_SCH1".MatCard[1, 2])
      R_Coil( "HMI_CMD_SCH1".Commands.MatCard.ResParts."8" )
   END_RUNG
   RUNG wire#powerrail
      Contact( "HMI_CMD_SCH1".Commands.MatCard.ResParts."9" )
      "MTS_Clear"(XS_MatCard := "STATUS_SCH1".MatCard[2, 2])
      R_Coil( "HMI_CMD_SCH1".Commands.MatCard.ResParts."9" )
   END_RUNG
   RUNG wire#powerrail
      Contact( "HMI_CMD_SCH1".Commands.MatCard.ResParts."10" )
      "MTS_Clear"(XS_MatCard := "STATUS_SCH1".MatCard[3, 2])
      R_Coil( "HMI_CMD_SCH1".Commands.MatCard.ResParts."10" )
   END_RUNG
   RUNG wire#powerrail
      Contact( "HMI_CMD_SCH1".Commands.MatCard.ResParts."11" )
      "MTS_Clear"(XS_MatCard := "STATUS_SCH1".MatCard[4, 2])
      R_Coil( "HMI_CMD_SCH1".Commands.MatCard.ResParts."11" )
   END_RUNG
   RUNG wire#powerrail
      Contact( "HMI_CMD_SCH1".Commands.MatCard.ResParts."12" )
      "MTS_Clear"(XS_MatCard := "STATUS_SCH1".MatCard[5, 2])
      R_Coil( "HMI_CMD_SCH1".Commands.MatCard.ResParts."12" )
   END_RUNG
   RUNG wire#powerrail
      Contact( "HMI_CMD_SCH1".Commands.MatCard.ResParts."13" )
      "MTS_Clear"(XS_MatCard := "STATUS_SCH1".MatCard[6, 2])
      R_Coil( "HMI_CMD_SCH1".Commands.MatCard.ResParts."13" )
   END_RUNG
   RUNG wire#powerrail
      Contact( "HMI_CMD_SCH1".Commands.MatCard.ResParts."14" )
      "MTS_Clear"(XS_MatCard := "STATUS_SCH1".MatCard[7, 2])
      R_Coil( "HMI_CMD_SCH1".Commands.MatCard.ResParts."14" )
   END_RUNG
   RUNG wire#powerrail
      Contact( "HMI_CMD_SCH1".Commands.MatCard.ResMap )
      "MTS_MapClear"(X_Map := "STATUS_SCH1".MatCard)
      R_Coil( "HMI_CMD_SCH1".Commands.MatCard.ResMap )
   END_RUNG
   // the same network as SCL:
   "MTS_Clear"(EN := "HMI_CMD_SCH1".Commands.MatCard.ResParts."1",
               XS_MatCard := "STATUS_SCH1".MatCard[1, 1],
               ENO => #_w1);
   IF #_w1 THEN "HMI_CMD_SCH1".Commands.MatCard.ResParts."1" := FALSE; END_IF;
   "MTS_Clear"(EN := "HMI_CMD_SCH1".Commands.MatCard.ResParts."2",
               XS_MatCard := "STATUS_SCH1".MatCard[2, 1],
               ENO => #_w2);
   IF #_w2 THEN "HMI_CMD_SCH1".Commands.MatCard.ResParts."2" := FALSE; END_IF;
   "MTS_Clear"(EN := "HMI_CMD_SCH1".Commands.MatCard.ResParts."3",
               XS_MatCard := "STATUS_SCH1".MatCard[3, 1],
               ENO => #_w3);
   IF #_w3 THEN "HMI_CMD_SCH1".Commands.MatCard.ResParts."3" := FALSE; END_IF;
   "MTS_Clear"(EN := "HMI_CMD_SCH1".Commands.MatCard.ResParts."4",
               XS_MatCard := "STATUS_SCH1".MatCard[4, 1],
               ENO => #_w4);
   IF #_w4 THEN "HMI_CMD_SCH1".Commands.MatCard.ResParts."4" := FALSE; END_IF;
   "MTS_Clear"(EN := "HMI_CMD_SCH1".Commands.MatCard.ResParts."5",
               XS_MatCard := "STATUS_SCH1".MatCard[5, 1],
               ENO => #_w5);
   IF #_w5 THEN "HMI_CMD_SCH1".Commands.MatCard.ResParts."5" := FALSE; END_IF;
   "MTS_Clear"(EN := "HMI_CMD_SCH1".Commands.MatCard.ResParts."6",
               XS_MatCard := "STATUS_SCH1".MatCard[6, 1],
               ENO => #_w6);
   IF #_w6 THEN "HMI_CMD_SCH1".Commands.MatCard.ResParts."6" := FALSE; END_IF;
   "MTS_Clear"(EN := "HMI_CMD_SCH1".Commands.MatCard.ResParts."7",
               XS_MatCard := "STATUS_SCH1".MatCard[7, 1],
               ENO => #_w7);
   IF #_w7 THEN "HMI_CMD_SCH1".Commands.MatCard.ResParts."7" := FALSE; END_IF;
   "MTS_Clear"(EN := "HMI_CMD_SCH1".Commands.MatCard.ResParts."8",
               XS_MatCard := "STATUS_SCH1".MatCard[1, 2],
               ENO => #_w8);
   IF #_w8 THEN "HMI_CMD_SCH1".Commands.MatCard.ResParts."8" := FALSE; END_IF;
   "MTS_Clear"(EN := "HMI_CMD_SCH1".Commands.MatCard.ResParts."9",
               XS_MatCard := "STATUS_SCH1".MatCard[2, 2],
               ENO => #_w9);
   IF #_w9 THEN "HMI_CMD_SCH1".Commands.MatCard.ResParts."9" := FALSE; END_IF;
   "MTS_Clear"(EN := "HMI_CMD_SCH1".Commands.MatCard.ResParts."10",
               XS_MatCard := "STATUS_SCH1".MatCard[3, 2],
               ENO => #_w10);
   IF #_w10 THEN "HMI_CMD_SCH1".Commands.MatCard.ResParts."10" := FALSE; END_IF;
   "MTS_Clear"(EN := "HMI_CMD_SCH1".Commands.MatCard.ResParts."11",
               XS_MatCard := "STATUS_SCH1".MatCard[4, 2],
               ENO => #_w11);
   IF #_w11 THEN "HMI_CMD_SCH1".Commands.MatCard.ResParts."11" := FALSE; END_IF;
   "MTS_Clear"(EN := "HMI_CMD_SCH1".Commands.MatCard.ResParts."12",
               XS_MatCard := "STATUS_SCH1".MatCard[5, 2],
               ENO => #_w12);
   IF #_w12 THEN "HMI_CMD_SCH1".Commands.MatCard.ResParts."12" := FALSE; END_IF;
   "MTS_Clear"(EN := "HMI_CMD_SCH1".Commands.MatCard.ResParts."13",
               XS_MatCard := "STATUS_SCH1".MatCard[6, 2],
               ENO => #_w13);
   IF #_w13 THEN "HMI_CMD_SCH1".Commands.MatCard.ResParts."13" := FALSE; END_IF;
   "MTS_Clear"(EN := "HMI_CMD_SCH1".Commands.MatCard.ResParts."14",
               XS_MatCard := "STATUS_SCH1".MatCard[7, 2],
               ENO => #_w14);
   IF #_w14 THEN "HMI_CMD_SCH1".Commands.MatCard.ResParts."14" := FALSE; END_IF;
   "MTS_MapClear"(EN := "HMI_CMD_SCH1".Commands.MatCard.ResMap, X_Map := "STATUS_SCH1".MatCard, ENO => #_w15);
   IF #_w15 THEN "HMI_CMD_SCH1".Commands.MatCard.ResMap := FALSE; END_IF;
END_REGION

REGION Network 28: Set positions in press - init
   // "JSA0Comm" - change when recipes done
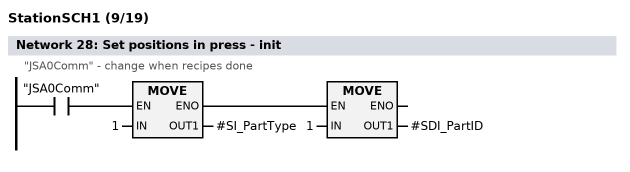
   RUNG wire#powerrail
      Contact( "JSA0Comm" )
      Move(in := 1, out1 => #SI_PartType)
      Move(in := 1, out1 => #SDI_PartID)
   END_RUNG
   // the same network as SCL:
   IF "JSA0Comm" THEN
       #SI_PartType := 1;
       #SDI_PartID := 1;
   END_IF;
END_REGION

REGION Network 29: Set positions in press - commands
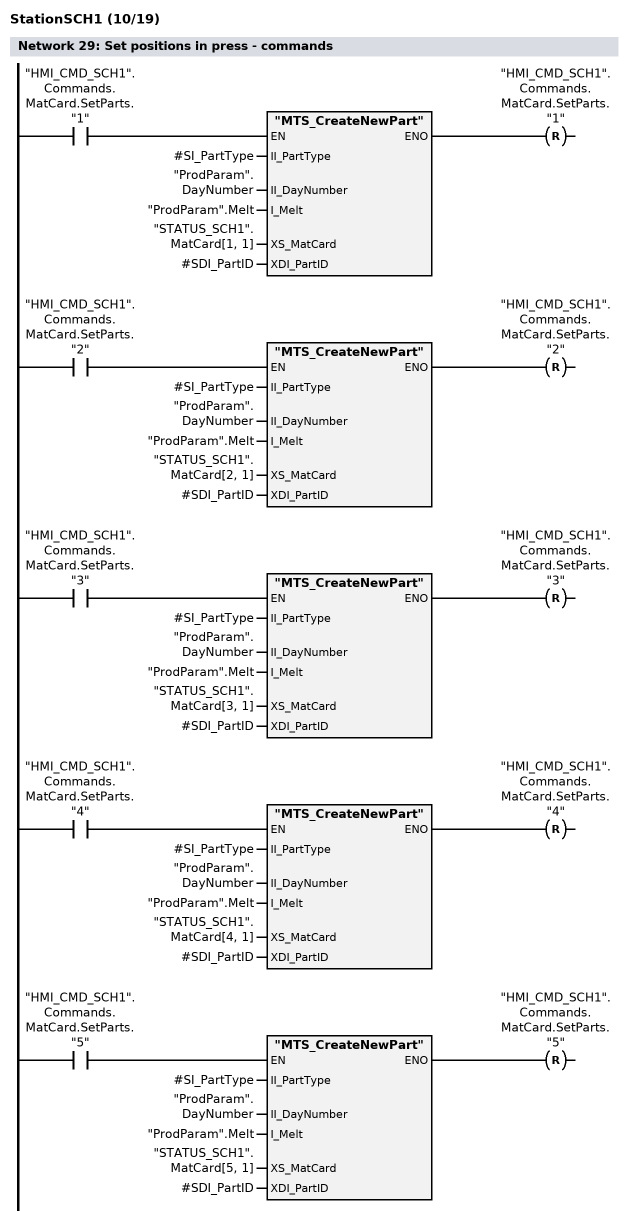
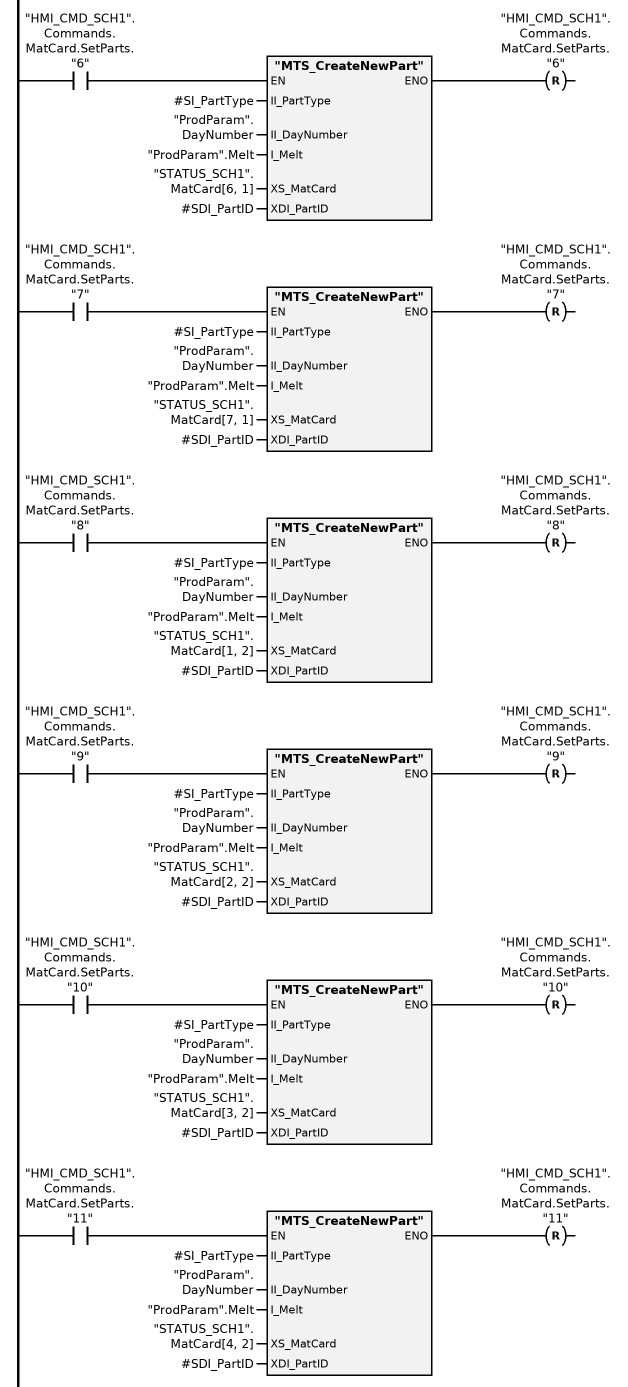
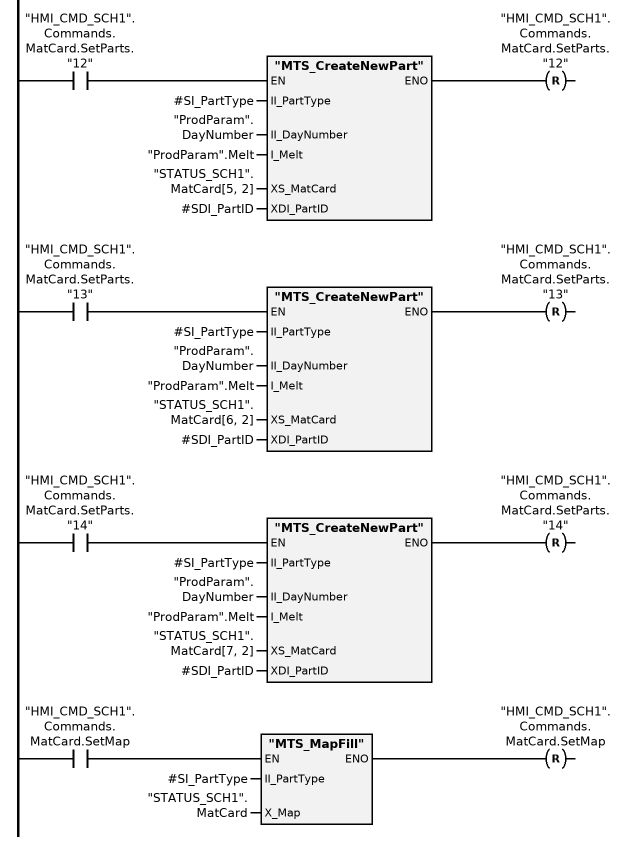
   RUNG wire#powerrail
      Contact( "HMI_CMD_SCH1".Commands.MatCard.SetParts."1" )
      "MTS_CreateNewPart"(II_PartType := #SI_PartType, II_DayNumber := "ProdParam".DayNumber, I_Melt := "ProdParam".Melt, XS_MatCard := "STATUS_SCH1".MatCard[1, 1], XDI_PartID := #SDI_PartID)
      R_Coil( "HMI_CMD_SCH1".Commands.MatCard.SetParts."1" )
   END_RUNG
   RUNG wire#powerrail
      Contact( "HMI_CMD_SCH1".Commands.MatCard.SetParts."2" )
      "MTS_CreateNewPart"(II_PartType := #SI_PartType, II_DayNumber := "ProdParam".DayNumber, I_Melt := "ProdParam".Melt, XS_MatCard := "STATUS_SCH1".MatCard[2, 1], XDI_PartID := #SDI_PartID)
      R_Coil( "HMI_CMD_SCH1".Commands.MatCard.SetParts."2" )
   END_RUNG
   RUNG wire#powerrail
      Contact( "HMI_CMD_SCH1".Commands.MatCard.SetParts."3" )
      "MTS_CreateNewPart"(II_PartType := #SI_PartType, II_DayNumber := "ProdParam".DayNumber, I_Melt := "ProdParam".Melt, XS_MatCard := "STATUS_SCH1".MatCard[3, 1], XDI_PartID := #SDI_PartID)
      R_Coil( "HMI_CMD_SCH1".Commands.MatCard.SetParts."3" )
   END_RUNG
   RUNG wire#powerrail
      Contact( "HMI_CMD_SCH1".Commands.MatCard.SetParts."4" )
      "MTS_CreateNewPart"(II_PartType := #SI_PartType, II_DayNumber := "ProdParam".DayNumber, I_Melt := "ProdParam".Melt, XS_MatCard := "STATUS_SCH1".MatCard[4, 1], XDI_PartID := #SDI_PartID)
      R_Coil( "HMI_CMD_SCH1".Commands.MatCard.SetParts."4" )
   END_RUNG
   RUNG wire#powerrail
      Contact( "HMI_CMD_SCH1".Commands.MatCard.SetParts."5" )
      "MTS_CreateNewPart"(II_PartType := #SI_PartType, II_DayNumber := "ProdParam".DayNumber, I_Melt := "ProdParam".Melt, XS_MatCard := "STATUS_SCH1".MatCard[5, 1], XDI_PartID := #SDI_PartID)
      R_Coil( "HMI_CMD_SCH1".Commands.MatCard.SetParts."5" )
   END_RUNG
   RUNG wire#powerrail
      Contact( "HMI_CMD_SCH1".Commands.MatCard.SetParts."6" )
      "MTS_CreateNewPart"(II_PartType := #SI_PartType, II_DayNumber := "ProdParam".DayNumber, I_Melt := "ProdParam".Melt, XS_MatCard := "STATUS_SCH1".MatCard[6, 1], XDI_PartID := #SDI_PartID)
      R_Coil( "HMI_CMD_SCH1".Commands.MatCard.SetParts."6" )
   END_RUNG
   RUNG wire#powerrail
      Contact( "HMI_CMD_SCH1".Commands.MatCard.SetParts."7" )
      "MTS_CreateNewPart"(II_PartType := #SI_PartType, II_DayNumber := "ProdParam".DayNumber, I_Melt := "ProdParam".Melt, XS_MatCard := "STATUS_SCH1".MatCard[7, 1], XDI_PartID := #SDI_PartID)
      R_Coil( "HMI_CMD_SCH1".Commands.MatCard.SetParts."7" )
   END_RUNG
   RUNG wire#powerrail
      Contact( "HMI_CMD_SCH1".Commands.MatCard.SetParts."8" )
      "MTS_CreateNewPart"(II_PartType := #SI_PartType, II_DayNumber := "ProdParam".DayNumber, I_Melt := "ProdParam".Melt, XS_MatCard := "STATUS_SCH1".MatCard[1, 2], XDI_PartID := #SDI_PartID)
      R_Coil( "HMI_CMD_SCH1".Commands.MatCard.SetParts."8" )
   END_RUNG
   RUNG wire#powerrail
      Contact( "HMI_CMD_SCH1".Commands.MatCard.SetParts."9" )
      "MTS_CreateNewPart"(II_PartType := #SI_PartType, II_DayNumber := "ProdParam".DayNumber, I_Melt := "ProdParam".Melt, XS_MatCard := "STATUS_SCH1".MatCard[2, 2], XDI_PartID := #SDI_PartID)
      R_Coil( "HMI_CMD_SCH1".Commands.MatCard.SetParts."9" )
   END_RUNG
   RUNG wire#powerrail
      Contact( "HMI_CMD_SCH1".Commands.MatCard.SetParts."10" )
      "MTS_CreateNewPart"(II_PartType := #SI_PartType, II_DayNumber := "ProdParam".DayNumber, I_Melt := "ProdParam".Melt, XS_MatCard := "STATUS_SCH1".MatCard[3, 2], XDI_PartID := #SDI_PartID)
      R_Coil( "HMI_CMD_SCH1".Commands.MatCard.SetParts."10" )
   END_RUNG
   RUNG wire#powerrail
      Contact( "HMI_CMD_SCH1".Commands.MatCard.SetParts."11" )
      "MTS_CreateNewPart"(II_PartType := #SI_PartType, II_DayNumber := "ProdParam".DayNumber, I_Melt := "ProdParam".Melt, XS_MatCard := "STATUS_SCH1".MatCard[4, 2], XDI_PartID := #SDI_PartID)
      R_Coil( "HMI_CMD_SCH1".Commands.MatCard.SetParts."11" )
   END_RUNG
   RUNG wire#powerrail
      Contact( "HMI_CMD_SCH1".Commands.MatCard.SetParts."12" )
      "MTS_CreateNewPart"(II_PartType := #SI_PartType, II_DayNumber := "ProdParam".DayNumber, I_Melt := "ProdParam".Melt, XS_MatCard := "STATUS_SCH1".MatCard[5, 2], XDI_PartID := #SDI_PartID)
      R_Coil( "HMI_CMD_SCH1".Commands.MatCard.SetParts."12" )
   END_RUNG
   RUNG wire#powerrail
      Contact( "HMI_CMD_SCH1".Commands.MatCard.SetParts."13" )
      "MTS_CreateNewPart"(II_PartType := #SI_PartType, II_DayNumber := "ProdParam".DayNumber, I_Melt := "ProdParam".Melt, XS_MatCard := "STATUS_SCH1".MatCard[6, 2], XDI_PartID := #SDI_PartID)
      R_Coil( "HMI_CMD_SCH1".Commands.MatCard.SetParts."13" )
   END_RUNG
   RUNG wire#powerrail
      Contact( "HMI_CMD_SCH1".Commands.MatCard.SetParts."14" )
      "MTS_CreateNewPart"(II_PartType := #SI_PartType, II_DayNumber := "ProdParam".DayNumber, I_Melt := "ProdParam".Melt, XS_MatCard := "STATUS_SCH1".MatCard[7, 2], XDI_PartID := #SDI_PartID)
      R_Coil( "HMI_CMD_SCH1".Commands.MatCard.SetParts."14" )
   END_RUNG
   RUNG wire#powerrail
      Contact( "HMI_CMD_SCH1".Commands.MatCard.SetMap )
      "MTS_MapFill"(II_PartType := #SI_PartType, X_Map := "STATUS_SCH1".MatCard)
      R_Coil( "HMI_CMD_SCH1".Commands.MatCard.SetMap )
   END_RUNG
   // the same network as SCL:
   "MTS_CreateNewPart"(EN := "HMI_CMD_SCH1".Commands.MatCard.SetParts."1",
                       II_PartType := #SI_PartType,
                       II_DayNumber := "ProdParam".DayNumber,
                       I_Melt := "ProdParam".Melt,
                       XS_MatCard := "STATUS_SCH1".MatCard[1, 1],
                       XDI_PartID := #SDI_PartID,
                       ENO => #_w1);
   IF #_w1 THEN "HMI_CMD_SCH1".Commands.MatCard.SetParts."1" := FALSE; END_IF;
   "MTS_CreateNewPart"(EN := "HMI_CMD_SCH1".Commands.MatCard.SetParts."2",
                       II_PartType := #SI_PartType,
                       II_DayNumber := "ProdParam".DayNumber,
                       I_Melt := "ProdParam".Melt,
                       XS_MatCard := "STATUS_SCH1".MatCard[2, 1],
                       XDI_PartID := #SDI_PartID,
                       ENO => #_w2);
   IF #_w2 THEN "HMI_CMD_SCH1".Commands.MatCard.SetParts."2" := FALSE; END_IF;
   "MTS_CreateNewPart"(EN := "HMI_CMD_SCH1".Commands.MatCard.SetParts."3",
                       II_PartType := #SI_PartType,
                       II_DayNumber := "ProdParam".DayNumber,
                       I_Melt := "ProdParam".Melt,
                       XS_MatCard := "STATUS_SCH1".MatCard[3, 1],
                       XDI_PartID := #SDI_PartID,
                       ENO => #_w3);
   IF #_w3 THEN "HMI_CMD_SCH1".Commands.MatCard.SetParts."3" := FALSE; END_IF;
   "MTS_CreateNewPart"(EN := "HMI_CMD_SCH1".Commands.MatCard.SetParts."4",
                       II_PartType := #SI_PartType,
                       II_DayNumber := "ProdParam".DayNumber,
                       I_Melt := "ProdParam".Melt,
                       XS_MatCard := "STATUS_SCH1".MatCard[4, 1],
                       XDI_PartID := #SDI_PartID,
                       ENO => #_w4);
   IF #_w4 THEN "HMI_CMD_SCH1".Commands.MatCard.SetParts."4" := FALSE; END_IF;
   "MTS_CreateNewPart"(EN := "HMI_CMD_SCH1".Commands.MatCard.SetParts."5",
                       II_PartType := #SI_PartType,
                       II_DayNumber := "ProdParam".DayNumber,
                       I_Melt := "ProdParam".Melt,
                       XS_MatCard := "STATUS_SCH1".MatCard[5, 1],
                       XDI_PartID := #SDI_PartID,
                       ENO => #_w5);
   IF #_w5 THEN "HMI_CMD_SCH1".Commands.MatCard.SetParts."5" := FALSE; END_IF;
   "MTS_CreateNewPart"(EN := "HMI_CMD_SCH1".Commands.MatCard.SetParts."6",
                       II_PartType := #SI_PartType,
                       II_DayNumber := "ProdParam".DayNumber,
                       I_Melt := "ProdParam".Melt,
                       XS_MatCard := "STATUS_SCH1".MatCard[6, 1],
                       XDI_PartID := #SDI_PartID,
                       ENO => #_w6);
   IF #_w6 THEN "HMI_CMD_SCH1".Commands.MatCard.SetParts."6" := FALSE; END_IF;
   "MTS_CreateNewPart"(EN := "HMI_CMD_SCH1".Commands.MatCard.SetParts."7",
                       II_PartType := #SI_PartType,
                       II_DayNumber := "ProdParam".DayNumber,
                       I_Melt := "ProdParam".Melt,
                       XS_MatCard := "STATUS_SCH1".MatCard[7, 1],
                       XDI_PartID := #SDI_PartID,
                       ENO => #_w7);
   IF #_w7 THEN "HMI_CMD_SCH1".Commands.MatCard.SetParts."7" := FALSE; END_IF;
   "MTS_CreateNewPart"(EN := "HMI_CMD_SCH1".Commands.MatCard.SetParts."8",
                       II_PartType := #SI_PartType,
                       II_DayNumber := "ProdParam".DayNumber,
                       I_Melt := "ProdParam".Melt,
                       XS_MatCard := "STATUS_SCH1".MatCard[1, 2],
                       XDI_PartID := #SDI_PartID,
                       ENO => #_w8);
   IF #_w8 THEN "HMI_CMD_SCH1".Commands.MatCard.SetParts."8" := FALSE; END_IF;
   "MTS_CreateNewPart"(EN := "HMI_CMD_SCH1".Commands.MatCard.SetParts."9",
                       II_PartType := #SI_PartType,
                       II_DayNumber := "ProdParam".DayNumber,
                       I_Melt := "ProdParam".Melt,
                       XS_MatCard := "STATUS_SCH1".MatCard[2, 2],
                       XDI_PartID := #SDI_PartID,
                       ENO => #_w9);
   IF #_w9 THEN "HMI_CMD_SCH1".Commands.MatCard.SetParts."9" := FALSE; END_IF;
   "MTS_CreateNewPart"(EN := "HMI_CMD_SCH1".Commands.MatCard.SetParts."10",
                       II_PartType := #SI_PartType,
                       II_DayNumber := "ProdParam".DayNumber,
                       I_Melt := "ProdParam".Melt,
                       XS_MatCard := "STATUS_SCH1".MatCard[3, 2],
                       XDI_PartID := #SDI_PartID,
                       ENO => #_w10);
   IF #_w10 THEN "HMI_CMD_SCH1".Commands.MatCard.SetParts."10" := FALSE; END_IF;
   "MTS_CreateNewPart"(EN := "HMI_CMD_SCH1".Commands.MatCard.SetParts."11",
                       II_PartType := #SI_PartType,
                       II_DayNumber := "ProdParam".DayNumber,
                       I_Melt := "ProdParam".Melt,
                       XS_MatCard := "STATUS_SCH1".MatCard[4, 2],
                       XDI_PartID := #SDI_PartID,
                       ENO => #_w11);
   IF #_w11 THEN "HMI_CMD_SCH1".Commands.MatCard.SetParts."11" := FALSE; END_IF;
   "MTS_CreateNewPart"(EN := "HMI_CMD_SCH1".Commands.MatCard.SetParts."12",
                       II_PartType := #SI_PartType,
                       II_DayNumber := "ProdParam".DayNumber,
                       I_Melt := "ProdParam".Melt,
                       XS_MatCard := "STATUS_SCH1".MatCard[5, 2],
                       XDI_PartID := #SDI_PartID,
                       ENO => #_w12);
   IF #_w12 THEN "HMI_CMD_SCH1".Commands.MatCard.SetParts."12" := FALSE; END_IF;
   "MTS_CreateNewPart"(EN := "HMI_CMD_SCH1".Commands.MatCard.SetParts."13",
                       II_PartType := #SI_PartType,
                       II_DayNumber := "ProdParam".DayNumber,
                       I_Melt := "ProdParam".Melt,
                       XS_MatCard := "STATUS_SCH1".MatCard[6, 2],
                       XDI_PartID := #SDI_PartID,
                       ENO => #_w13);
   IF #_w13 THEN "HMI_CMD_SCH1".Commands.MatCard.SetParts."13" := FALSE; END_IF;
   "MTS_CreateNewPart"(EN := "HMI_CMD_SCH1".Commands.MatCard.SetParts."14",
                       II_PartType := #SI_PartType,
                       II_DayNumber := "ProdParam".DayNumber,
                       I_Melt := "ProdParam".Melt,
                       XS_MatCard := "STATUS_SCH1".MatCard[7, 2],
                       XDI_PartID := #SDI_PartID,
                       ENO => #_w14);
   IF #_w14 THEN "HMI_CMD_SCH1".Commands.MatCard.SetParts."14" := FALSE; END_IF;
   "MTS_MapFill"(EN := "HMI_CMD_SCH1".Commands.MatCard.SetMap,
                 II_PartType := #SI_PartType,
                 X_Map := "STATUS_SCH1".MatCard,
                 ENO => #_w15);
   IF #_w15 THEN "HMI_CMD_SCH1".Commands.MatCard.SetMap := FALSE; END_IF;
END_REGION

REGION Network 30: Data transfer: Press die 7 (cutting) -> Output conveyor (BSN3 infeed)
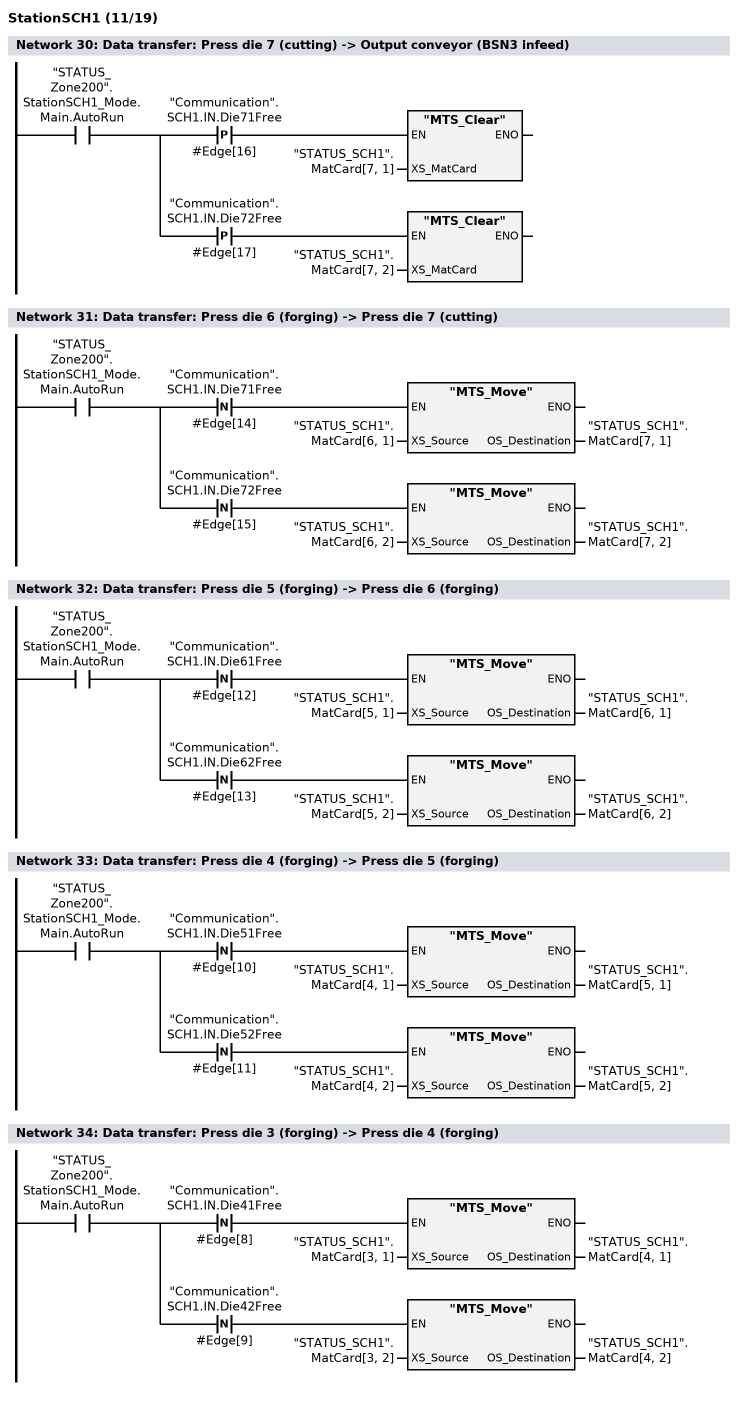
   RUNG wire#powerrail
      Contact( "STATUS_Zone200".StationSCH1_Mode.Main.AutoRun )
      wire#w1
      P_Contact(operand := "Communication".SCH1.IN.Die71Free, bit := #Edge[16])
      "MTS_Clear"(XS_MatCard := "STATUS_SCH1".MatCard[7, 1])
   END_RUNG
   RUNG wire#w1
      P_Contact(operand := "Communication".SCH1.IN.Die72Free, bit := #Edge[17])
      "MTS_Clear"(XS_MatCard := "STATUS_SCH1".MatCard[7, 2])
   END_RUNG
   // the same network as SCL:
   #_w1 := "STATUS_Zone200".StationSCH1_Mode.Main.AutoRun AND "Communication".SCH1.IN.Die71Free AND NOT #Edge[16];   // rising edge of "Communication".SCH1.IN.Die71Free
   #Edge[16] := "Communication".SCH1.IN.Die71Free;
   #_w2 := "STATUS_Zone200".StationSCH1_Mode.Main.AutoRun;
   IF #_w1 THEN "MTS_Clear"(XS_MatCard := "STATUS_SCH1".MatCard[7, 1]); END_IF;
   #_w3 := #_w2 AND "Communication".SCH1.IN.Die72Free AND NOT #Edge[17];   // rising edge of "Communication".SCH1.IN.Die72Free
   #Edge[17] := "Communication".SCH1.IN.Die72Free;
   IF #_w3 THEN "MTS_Clear"(XS_MatCard := "STATUS_SCH1".MatCard[7, 2]); END_IF;
END_REGION

REGION Network 31: Data transfer: Press die 6 (forging) -> Press die 7 (cutting)
   RUNG wire#powerrail
      Contact( "STATUS_Zone200".StationSCH1_Mode.Main.AutoRun )
      wire#w1
      N_Contact(operand := "Communication".SCH1.IN.Die71Free, bit := #Edge[14])
      "MTS_Move"(XS_Source := "STATUS_SCH1".MatCard[6, 1], OS_Destination => "STATUS_SCH1".MatCard[7, 1])
   END_RUNG
   RUNG wire#w1
      N_Contact(operand := "Communication".SCH1.IN.Die72Free, bit := #Edge[15])
      "MTS_Move"(XS_Source := "STATUS_SCH1".MatCard[6, 2], OS_Destination => "STATUS_SCH1".MatCard[7, 2])
   END_RUNG
   // the same network as SCL:
   #_w1 := "STATUS_Zone200".StationSCH1_Mode.Main.AutoRun AND NOT "Communication".SCH1.IN.Die71Free AND #Edge[14];   // falling edge of "Communication".SCH1.IN.Die71Free
   #Edge[14] := "Communication".SCH1.IN.Die71Free;
   #_w2 := "STATUS_Zone200".StationSCH1_Mode.Main.AutoRun;
   IF #_w1 THEN
       "MTS_Move"(XS_Source := "STATUS_SCH1".MatCard[6, 1], OS_Destination => "STATUS_SCH1".MatCard[7, 1]);
   END_IF;
   #_w3 := #_w2 AND NOT "Communication".SCH1.IN.Die72Free AND #Edge[15];   // falling edge of "Communication".SCH1.IN.Die72Free
   #Edge[15] := "Communication".SCH1.IN.Die72Free;
   IF #_w3 THEN
       "MTS_Move"(XS_Source := "STATUS_SCH1".MatCard[6, 2], OS_Destination => "STATUS_SCH1".MatCard[7, 2]);
   END_IF;
END_REGION

REGION Network 32: Data transfer: Press die 5 (forging) -> Press die 6 (forging)
   RUNG wire#powerrail
      Contact( "STATUS_Zone200".StationSCH1_Mode.Main.AutoRun )
      wire#w1
      N_Contact(operand := "Communication".SCH1.IN.Die61Free, bit := #Edge[12])
      "MTS_Move"(XS_Source := "STATUS_SCH1".MatCard[5, 1], OS_Destination => "STATUS_SCH1".MatCard[6, 1])
   END_RUNG
   RUNG wire#w1
      N_Contact(operand := "Communication".SCH1.IN.Die62Free, bit := #Edge[13])
      "MTS_Move"(XS_Source := "STATUS_SCH1".MatCard[5, 2], OS_Destination => "STATUS_SCH1".MatCard[6, 2])
   END_RUNG
   // the same network as SCL:
   #_w1 := "STATUS_Zone200".StationSCH1_Mode.Main.AutoRun AND NOT "Communication".SCH1.IN.Die61Free AND #Edge[12];   // falling edge of "Communication".SCH1.IN.Die61Free
   #Edge[12] := "Communication".SCH1.IN.Die61Free;
   #_w2 := "STATUS_Zone200".StationSCH1_Mode.Main.AutoRun;
   IF #_w1 THEN
       "MTS_Move"(XS_Source := "STATUS_SCH1".MatCard[5, 1], OS_Destination => "STATUS_SCH1".MatCard[6, 1]);
   END_IF;
   #_w3 := #_w2 AND NOT "Communication".SCH1.IN.Die62Free AND #Edge[13];   // falling edge of "Communication".SCH1.IN.Die62Free
   #Edge[13] := "Communication".SCH1.IN.Die62Free;
   IF #_w3 THEN
       "MTS_Move"(XS_Source := "STATUS_SCH1".MatCard[5, 2], OS_Destination => "STATUS_SCH1".MatCard[6, 2]);
   END_IF;
END_REGION

REGION Network 33: Data transfer: Press die 4 (forging) -> Press die 5 (forging)
   RUNG wire#powerrail
      Contact( "STATUS_Zone200".StationSCH1_Mode.Main.AutoRun )
      wire#w1
      N_Contact(operand := "Communication".SCH1.IN.Die51Free, bit := #Edge[10])
      "MTS_Move"(XS_Source := "STATUS_SCH1".MatCard[4, 1], OS_Destination => "STATUS_SCH1".MatCard[5, 1])
   END_RUNG
   RUNG wire#w1
      N_Contact(operand := "Communication".SCH1.IN.Die52Free, bit := #Edge[11])
      "MTS_Move"(XS_Source := "STATUS_SCH1".MatCard[4, 2], OS_Destination => "STATUS_SCH1".MatCard[5, 2])
   END_RUNG
   // the same network as SCL:
   #_w1 := "STATUS_Zone200".StationSCH1_Mode.Main.AutoRun AND NOT "Communication".SCH1.IN.Die51Free AND #Edge[10];   // falling edge of "Communication".SCH1.IN.Die51Free
   #Edge[10] := "Communication".SCH1.IN.Die51Free;
   #_w2 := "STATUS_Zone200".StationSCH1_Mode.Main.AutoRun;
   IF #_w1 THEN
       "MTS_Move"(XS_Source := "STATUS_SCH1".MatCard[4, 1], OS_Destination => "STATUS_SCH1".MatCard[5, 1]);
   END_IF;
   #_w3 := #_w2 AND NOT "Communication".SCH1.IN.Die52Free AND #Edge[11];   // falling edge of "Communication".SCH1.IN.Die52Free
   #Edge[11] := "Communication".SCH1.IN.Die52Free;
   IF #_w3 THEN
       "MTS_Move"(XS_Source := "STATUS_SCH1".MatCard[4, 2], OS_Destination => "STATUS_SCH1".MatCard[5, 2]);
   END_IF;
END_REGION

REGION Network 34: Data transfer: Press die 3 (forging) -> Press die 4 (forging)
   RUNG wire#powerrail
      Contact( "STATUS_Zone200".StationSCH1_Mode.Main.AutoRun )
      wire#w1
      N_Contact(operand := "Communication".SCH1.IN.Die41Free, bit := #Edge[8])
      "MTS_Move"(XS_Source := "STATUS_SCH1".MatCard[3, 1], OS_Destination => "STATUS_SCH1".MatCard[4, 1])
   END_RUNG
   RUNG wire#w1
      N_Contact(operand := "Communication".SCH1.IN.Die42Free, bit := #Edge[9])
      "MTS_Move"(XS_Source := "STATUS_SCH1".MatCard[3, 2], OS_Destination => "STATUS_SCH1".MatCard[4, 2])
   END_RUNG
   // the same network as SCL:
   #_w1 := "STATUS_Zone200".StationSCH1_Mode.Main.AutoRun AND NOT "Communication".SCH1.IN.Die41Free AND #Edge[8];   // falling edge of "Communication".SCH1.IN.Die41Free
   #Edge[8] := "Communication".SCH1.IN.Die41Free;
   #_w2 := "STATUS_Zone200".StationSCH1_Mode.Main.AutoRun;
   IF #_w1 THEN
       "MTS_Move"(XS_Source := "STATUS_SCH1".MatCard[3, 1], OS_Destination => "STATUS_SCH1".MatCard[4, 1]);
   END_IF;
   #_w3 := #_w2 AND NOT "Communication".SCH1.IN.Die42Free AND #Edge[9];   // falling edge of "Communication".SCH1.IN.Die42Free
   #Edge[9] := "Communication".SCH1.IN.Die42Free;
   IF #_w3 THEN
       "MTS_Move"(XS_Source := "STATUS_SCH1".MatCard[3, 2], OS_Destination => "STATUS_SCH1".MatCard[4, 2]);
   END_IF;
END_REGION

REGION Network 35: Data transfer: Press die 2 (buffer) -> Press die 3 (forging)
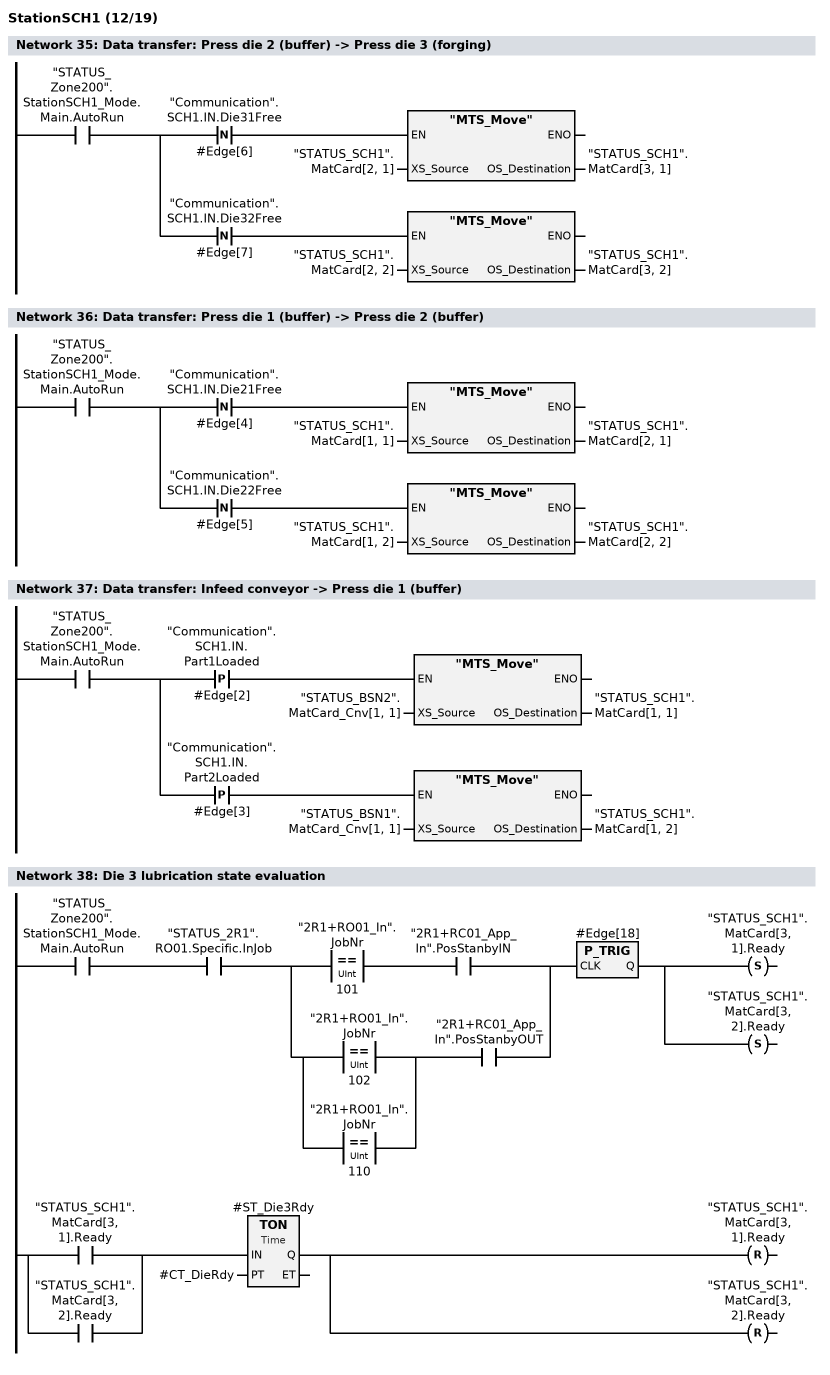
   RUNG wire#powerrail
      Contact( "STATUS_Zone200".StationSCH1_Mode.Main.AutoRun )
      wire#w1
      N_Contact(operand := "Communication".SCH1.IN.Die31Free, bit := #Edge[6])
      "MTS_Move"(XS_Source := "STATUS_SCH1".MatCard[2, 1], OS_Destination => "STATUS_SCH1".MatCard[3, 1])
   END_RUNG
   RUNG wire#w1
      N_Contact(operand := "Communication".SCH1.IN.Die32Free, bit := #Edge[7])
      "MTS_Move"(XS_Source := "STATUS_SCH1".MatCard[2, 2], OS_Destination => "STATUS_SCH1".MatCard[3, 2])
   END_RUNG
   // the same network as SCL:
   #_w1 := "STATUS_Zone200".StationSCH1_Mode.Main.AutoRun AND NOT "Communication".SCH1.IN.Die31Free AND #Edge[6];   // falling edge of "Communication".SCH1.IN.Die31Free
   #Edge[6] := "Communication".SCH1.IN.Die31Free;
   #_w2 := "STATUS_Zone200".StationSCH1_Mode.Main.AutoRun;
   IF #_w1 THEN
       "MTS_Move"(XS_Source := "STATUS_SCH1".MatCard[2, 1], OS_Destination => "STATUS_SCH1".MatCard[3, 1]);
   END_IF;
   #_w3 := #_w2 AND NOT "Communication".SCH1.IN.Die32Free AND #Edge[7];   // falling edge of "Communication".SCH1.IN.Die32Free
   #Edge[7] := "Communication".SCH1.IN.Die32Free;
   IF #_w3 THEN
       "MTS_Move"(XS_Source := "STATUS_SCH1".MatCard[2, 2], OS_Destination => "STATUS_SCH1".MatCard[3, 2]);
   END_IF;
END_REGION

REGION Network 36: Data transfer: Press die 1 (buffer) -> Press die 2 (buffer)
   RUNG wire#powerrail
      Contact( "STATUS_Zone200".StationSCH1_Mode.Main.AutoRun )
      wire#w1
      N_Contact(operand := "Communication".SCH1.IN.Die21Free, bit := #Edge[4])
      "MTS_Move"(XS_Source := "STATUS_SCH1".MatCard[1, 1], OS_Destination => "STATUS_SCH1".MatCard[2, 1])
   END_RUNG
   RUNG wire#w1
      N_Contact(operand := "Communication".SCH1.IN.Die22Free, bit := #Edge[5])
      "MTS_Move"(XS_Source := "STATUS_SCH1".MatCard[1, 2], OS_Destination => "STATUS_SCH1".MatCard[2, 2])
   END_RUNG
   // the same network as SCL:
   #_w1 := "STATUS_Zone200".StationSCH1_Mode.Main.AutoRun AND NOT "Communication".SCH1.IN.Die21Free AND #Edge[4];   // falling edge of "Communication".SCH1.IN.Die21Free
   #Edge[4] := "Communication".SCH1.IN.Die21Free;
   #_w2 := "STATUS_Zone200".StationSCH1_Mode.Main.AutoRun;
   IF #_w1 THEN
       "MTS_Move"(XS_Source := "STATUS_SCH1".MatCard[1, 1], OS_Destination => "STATUS_SCH1".MatCard[2, 1]);
   END_IF;
   #_w3 := #_w2 AND NOT "Communication".SCH1.IN.Die22Free AND #Edge[5];   // falling edge of "Communication".SCH1.IN.Die22Free
   #Edge[5] := "Communication".SCH1.IN.Die22Free;
   IF #_w3 THEN
       "MTS_Move"(XS_Source := "STATUS_SCH1".MatCard[1, 2], OS_Destination => "STATUS_SCH1".MatCard[2, 2]);
   END_IF;
END_REGION

REGION Network 37: Data transfer: Infeed conveyor -> Press die 1 (buffer)
   RUNG wire#powerrail
      Contact( "STATUS_Zone200".StationSCH1_Mode.Main.AutoRun )
      wire#w1
      P_Contact(operand := "Communication".SCH1.IN.Part1Loaded, bit := #Edge[2])
      "MTS_Move"(XS_Source := "STATUS_BSN2".MatCard_Cnv[1, 1], OS_Destination => "STATUS_SCH1".MatCard[1, 1])
   END_RUNG
   RUNG wire#w1
      P_Contact(operand := "Communication".SCH1.IN.Part2Loaded, bit := #Edge[3])
      "MTS_Move"(XS_Source := "STATUS_BSN1".MatCard_Cnv[1, 1], OS_Destination => "STATUS_SCH1".MatCard[1, 2])
   END_RUNG
   // the same network as SCL:
   #_w1 := "STATUS_Zone200".StationSCH1_Mode.Main.AutoRun AND "Communication".SCH1.IN.Part1Loaded AND NOT #Edge[2];   // rising edge of "Communication".SCH1.IN.Part1Loaded
   #Edge[2] := "Communication".SCH1.IN.Part1Loaded;
   #_w2 := "STATUS_Zone200".StationSCH1_Mode.Main.AutoRun;
   IF #_w1 THEN
       "MTS_Move"(XS_Source := "STATUS_BSN2".MatCard_Cnv[1, 1], OS_Destination => "STATUS_SCH1".MatCard[1, 1]);
   END_IF;
   #_w3 := #_w2 AND "Communication".SCH1.IN.Part2Loaded AND NOT #Edge[3];   // rising edge of "Communication".SCH1.IN.Part2Loaded
   #Edge[3] := "Communication".SCH1.IN.Part2Loaded;
   IF #_w3 THEN
       "MTS_Move"(XS_Source := "STATUS_BSN1".MatCard_Cnv[1, 1], OS_Destination => "STATUS_SCH1".MatCard[1, 2]);
   END_IF;
END_REGION

REGION Network 38: Die 3 lubrication state evaluation
   RUNG wire#powerrail
      Contact( "STATUS_Zone200".StationSCH1_Mode.Main.AutoRun )
      Contact( "STATUS_2R1".RO01.Specific.InJob )
      wire#w1
      { S7_Templates := "SrcType := UInt" } EQ_Contact(in1 := "2R1+RO01_In".JobNr, in2 := 101)
      Contact( "2R1+RC01_App_In".PosStanbyIN )
      wire#w2
      P_Trig( #Edge[18] )
      wire#w4
      S_Coil( "STATUS_SCH1".MatCard[3, 1].Ready )
   END_RUNG
   RUNG wire#w1
      { S7_Templates := "SrcType := UInt" } EQ_Contact(in1 := "2R1+RO01_In".JobNr, in2 := 102)
      wire#w3
      Contact( "2R1+RC01_App_In".PosStanbyOUT )
   END_RUNG wire#w2
   RUNG wire#w1
      { S7_Templates := "SrcType := UInt" } EQ_Contact(in1 := "2R1+RO01_In".JobNr, in2 := 110)
   END_RUNG wire#w3
   RUNG wire#w4
      S_Coil( "STATUS_SCH1".MatCard[3, 2].Ready )
   END_RUNG
   RUNG wire#powerrail
      Contact( "STATUS_SCH1".MatCard[3, 1].Ready )
      wire#w5
      { S7_Templates := "time_type := Time" } #ST_Die3Rdy.TON(pt := #CT_DieRdy, et =>)
      wire#w6
      R_Coil( "STATUS_SCH1".MatCard[3, 1].Ready )
   END_RUNG
   RUNG wire#powerrail
      Contact( "STATUS_SCH1".MatCard[3, 2].Ready )
   END_RUNG wire#w5
   RUNG wire#w6
      R_Coil( "STATUS_SCH1".MatCard[3, 2].Ready )
   END_RUNG
   // the same network as SCL:
   #_w1 := "STATUS_Zone200".StationSCH1_Mode.Main.AutoRun AND "STATUS_2R1".RO01.Specific.InJob AND ((("2R1+RO01_In".JobNr = 101) AND "2R1+RC01_App_In".PosStanbyIN) OR ((("2R1+RO01_In".JobNr = 102) OR ("2R1+RO01_In".JobNr = 110)) AND "2R1+RC01_App_In".PosStanbyOUT));
   #_w2 := #_w1 AND NOT #Edge[18];   // rising edge
   #Edge[18] := #_w1;
   IF #_w2 THEN
       "STATUS_SCH1".MatCard[3, 1].Ready := TRUE;
       "STATUS_SCH1".MatCard[3, 2].Ready := TRUE;
   END_IF;
   #ST_Die3Rdy(IN := "STATUS_SCH1".MatCard[3, 1].Ready OR "STATUS_SCH1".MatCard[3, 2].Ready, PT := #CT_DieRdy);   // TON
   IF #ST_Die3Rdy.Q THEN
       "STATUS_SCH1".MatCard[3, 1].Ready := FALSE;
       "STATUS_SCH1".MatCard[3, 2].Ready := FALSE;
   END_IF;
END_REGION

REGION Network 39: Die 4, 5, 6 lubrication state evaluation
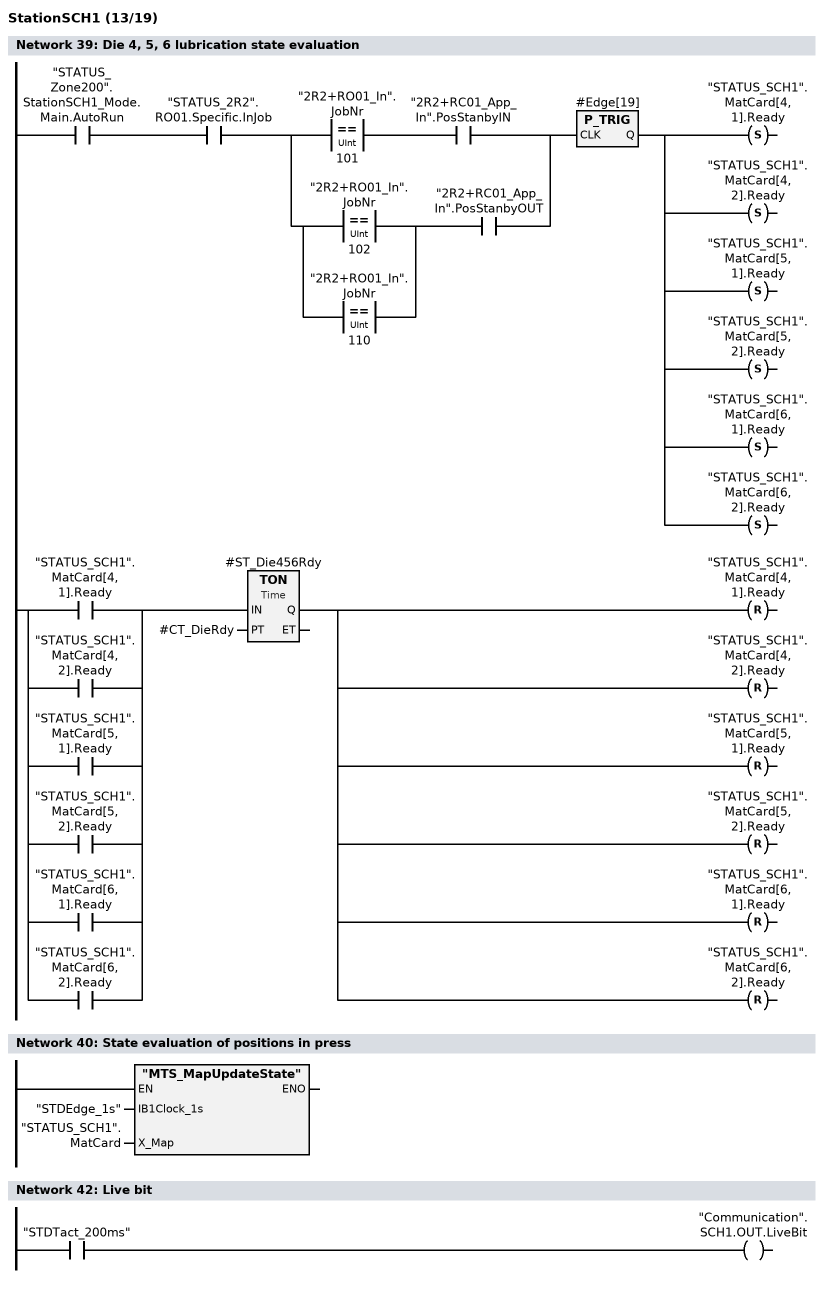
   RUNG wire#powerrail
      Contact( "STATUS_Zone200".StationSCH1_Mode.Main.AutoRun )
      Contact( "STATUS_2R2".RO01.Specific.InJob )
      wire#w1
      { S7_Templates := "SrcType := UInt" } EQ_Contact(in1 := "2R2+RO01_In".JobNr, in2 := 101)
      Contact( "2R2+RC01_App_In".PosStanbyIN )
      wire#w2
      P_Trig( #Edge[19] )
      wire#w4
      S_Coil( "STATUS_SCH1".MatCard[4, 1].Ready )
   END_RUNG
   RUNG wire#w1
      { S7_Templates := "SrcType := UInt" } EQ_Contact(in1 := "2R2+RO01_In".JobNr, in2 := 102)
      wire#w3
      Contact( "2R2+RC01_App_In".PosStanbyOUT )
   END_RUNG wire#w2
   RUNG wire#w1
      { S7_Templates := "SrcType := UInt" } EQ_Contact(in1 := "2R2+RO01_In".JobNr, in2 := 110)
   END_RUNG wire#w3
   RUNG wire#w4
      S_Coil( "STATUS_SCH1".MatCard[4, 2].Ready )
   END_RUNG
   RUNG wire#w4
      S_Coil( "STATUS_SCH1".MatCard[5, 1].Ready )
   END_RUNG
   RUNG wire#w4
      S_Coil( "STATUS_SCH1".MatCard[5, 2].Ready )
   END_RUNG
   RUNG wire#w4
      S_Coil( "STATUS_SCH1".MatCard[6, 1].Ready )
   END_RUNG
   RUNG wire#w4
      S_Coil( "STATUS_SCH1".MatCard[6, 2].Ready )
   END_RUNG
   RUNG wire#powerrail
      Contact( "STATUS_SCH1".MatCard[4, 1].Ready )
      wire#w5
      { S7_Templates := "time_type := Time" } #ST_Die456Rdy.TON(pt := #CT_DieRdy, et =>)
      wire#w6
      R_Coil( "STATUS_SCH1".MatCard[4, 1].Ready )
   END_RUNG
   RUNG wire#powerrail
      Contact( "STATUS_SCH1".MatCard[4, 2].Ready )
   END_RUNG wire#w5
   RUNG wire#powerrail
      Contact( "STATUS_SCH1".MatCard[5, 1].Ready )
   END_RUNG wire#w5
   RUNG wire#powerrail
      Contact( "STATUS_SCH1".MatCard[5, 2].Ready )
   END_RUNG wire#w5
   RUNG wire#powerrail
      Contact( "STATUS_SCH1".MatCard[6, 1].Ready )
   END_RUNG wire#w5
   RUNG wire#powerrail
      Contact( "STATUS_SCH1".MatCard[6, 2].Ready )
   END_RUNG wire#w5
   RUNG wire#w6
      R_Coil( "STATUS_SCH1".MatCard[4, 2].Ready )
   END_RUNG
   RUNG wire#w6
      R_Coil( "STATUS_SCH1".MatCard[5, 1].Ready )
   END_RUNG
   RUNG wire#w6
      R_Coil( "STATUS_SCH1".MatCard[5, 2].Ready )
   END_RUNG
   RUNG wire#w6
      R_Coil( "STATUS_SCH1".MatCard[6, 1].Ready )
   END_RUNG
   RUNG wire#w6
      R_Coil( "STATUS_SCH1".MatCard[6, 2].Ready )
   END_RUNG
   // the same network as SCL:
   #_w1 := "STATUS_Zone200".StationSCH1_Mode.Main.AutoRun AND "STATUS_2R2".RO01.Specific.InJob AND ((("2R2+RO01_In".JobNr = 101) AND "2R2+RC01_App_In".PosStanbyIN) OR ((("2R2+RO01_In".JobNr = 102) OR ("2R2+RO01_In".JobNr = 110)) AND "2R2+RC01_App_In".PosStanbyOUT));
   #_w2 := #_w1 AND NOT #Edge[19];   // rising edge
   #Edge[19] := #_w1;
   IF #_w2 THEN
       "STATUS_SCH1".MatCard[4, 1].Ready := TRUE;
       "STATUS_SCH1".MatCard[4, 2].Ready := TRUE;
       "STATUS_SCH1".MatCard[5, 1].Ready := TRUE;
       "STATUS_SCH1".MatCard[5, 2].Ready := TRUE;
       "STATUS_SCH1".MatCard[6, 1].Ready := TRUE;
       "STATUS_SCH1".MatCard[6, 2].Ready := TRUE;
   END_IF;
   #ST_Die456Rdy(IN := "STATUS_SCH1".MatCard[4, 1].Ready OR "STATUS_SCH1".MatCard[4, 2].Ready OR "STATUS_SCH1".MatCard[5, 1].Ready OR "STATUS_SCH1".MatCard[5, 2].Ready OR "STATUS_SCH1".MatCard[6, 1].Ready OR "STATUS_SCH1".MatCard[6, 2].Ready,   // TON
                 PT := #CT_DieRdy);
   IF #ST_Die456Rdy.Q THEN
       "STATUS_SCH1".MatCard[4, 1].Ready := FALSE;
       "STATUS_SCH1".MatCard[4, 2].Ready := FALSE;
       "STATUS_SCH1".MatCard[5, 1].Ready := FALSE;
       "STATUS_SCH1".MatCard[5, 2].Ready := FALSE;
       "STATUS_SCH1".MatCard[6, 1].Ready := FALSE;
       "STATUS_SCH1".MatCard[6, 2].Ready := FALSE;
   END_IF;
END_REGION

REGION Network 40: State evaluation of positions in press
   RUNG wire#powerrail
      "MTS_MapUpdateState"(IB1Clock_1s := "STDEdge_1s", X_Map := "STATUS_SCH1".MatCard)
   END_RUNG
   // the same network as SCL:
   "MTS_MapUpdateState"(IB1Clock_1s := "STDEdge_1s", X_Map := "STATUS_SCH1".MatCard);
END_REGION

REGION Network 41: *************** Interface to press machine ***************
END_REGION

REGION Network 42: Live bit
   RUNG wire#powerrail
      Contact( "STDTact_200ms" )
      Coil( "Communication".SCH1.OUT.LiveBit )
   END_RUNG
   // the same network as SCL:
   "Communication".SCH1.OUT.LiveBit := "STDTact_200ms";
END_REGION

REGION Network 43: Error acknowledge
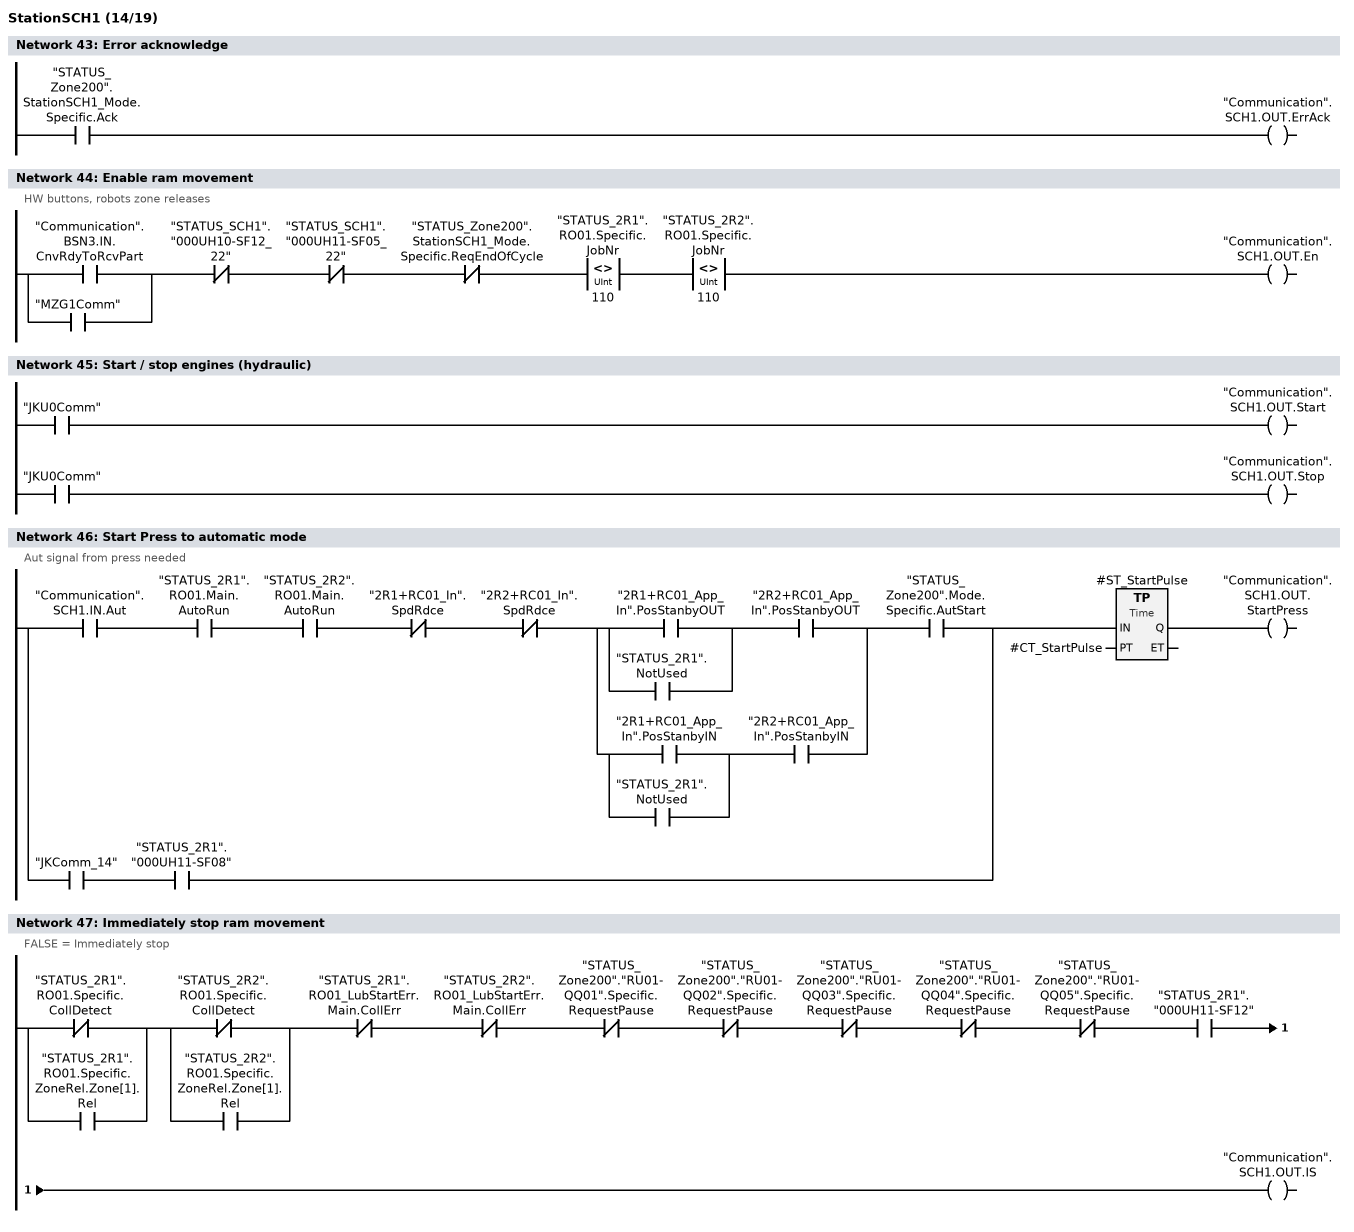
   RUNG wire#powerrail
      Contact( "STATUS_Zone200".StationSCH1_Mode.Specific.Ack )
      Coil( "Communication".SCH1.OUT.ErrAck )
   END_RUNG
   // the same network as SCL:
   "Communication".SCH1.OUT.ErrAck := "STATUS_Zone200".StationSCH1_Mode.Specific.Ack;
END_REGION

REGION Network 44: Enable ram movement
   // HW buttons, robots zone releases
   RUNG wire#powerrail
      Contact( "Communication".BSN3.IN.CnvRdyToRcvPart )
      wire#w1
      I_Contact( "STATUS_SCH1"."000UH10-SF12_22" )
      I_Contact( "STATUS_SCH1"."000UH11-SF05_22" )
      I_Contact( "STATUS_Zone200".StationSCH1_Mode.Specific.ReqEndOfCycle )
      { S7_Templates := "SrcType := UInt" } NE_Contact(in1 := "STATUS_2R1".RO01.Specific.JobNr, in2 := 110)
      { S7_Templates := "SrcType := UInt" } NE_Contact(in1 := "STATUS_2R2".RO01.Specific.JobNr, in2 := 110)
      Coil( "Communication".SCH1.OUT.En )
   END_RUNG
   RUNG wire#powerrail
      Contact( "MZG1Comm" )
   END_RUNG wire#w1
   // the same network as SCL:
   "Communication".SCH1.OUT.En := ("Communication".BSN3.IN.CnvRdyToRcvPart OR "MZG1Comm") AND NOT "STATUS_SCH1"."000UH10-SF12_22" AND NOT "STATUS_SCH1"."000UH11-SF05_22" AND NOT "STATUS_Zone200".StationSCH1_Mode.Specific.ReqEndOfCycle AND ("STATUS_2R1".RO01.Specific.JobNr <> 110) AND ("STATUS_2R2".RO01.Specific.JobNr <> 110);
END_REGION

REGION Network 45: Start / stop engines (hydraulic)
   RUNG wire#powerrail
      Contact( "JKU0Comm" )
      Coil( "Communication".SCH1.OUT.Start )
   END_RUNG
   RUNG wire#powerrail
      Contact( "JKU0Comm" )
      Coil( "Communication".SCH1.OUT.Stop )
   END_RUNG
   // the same network as SCL:
   "Communication".SCH1.OUT.Start := "JKU0Comm";
   "Communication".SCH1.OUT.Stop := "JKU0Comm";
END_REGION

REGION Network 46: Start Press to automatic mode
   // Aut signal from press needed
   RUNG wire#powerrail
      Contact( "Communication".SCH1.IN.Aut )
      Contact( "STATUS_2R1".RO01.Main.AutoRun )
      Contact( "STATUS_2R2".RO01.Main.AutoRun )
      I_Contact( "2R1+RC01_In".SpdRdce )
      I_Contact( "2R2+RC01_In".SpdRdce )
      wire#w1
      Contact( "2R1+RC01_App_In".PosStanbyOUT )
      wire#w2
      Contact( "2R2+RC01_App_In".PosStanbyOUT )
      wire#w3
      Contact( "STATUS_Zone200".Mode.Specific.AutStart )
      wire#w5
      { S7_Templates := "time_type := Time" } #ST_StartPulse.TP(pt := #CT_StartPulse, et =>)
      Coil( "Communication".SCH1.OUT.StartPress )
   END_RUNG
   RUNG wire#w1
      Contact( "STATUS_2R1".NotUsed )
   END_RUNG wire#w2
   RUNG wire#w1
      Contact( "2R1+RC01_App_In".PosStanbyIN )
      wire#w4
      Contact( "2R2+RC01_App_In".PosStanbyIN )
   END_RUNG wire#w3
   RUNG wire#w1
      Contact( "STATUS_2R1".NotUsed )
   END_RUNG wire#w4
   RUNG wire#powerrail
      Contact( "JKComm_14" )
      Contact( "STATUS_2R1"."000UH11-SF08" )
   END_RUNG wire#w5
   // the same network as SCL:
   #ST_StartPulse(IN := ("Communication".SCH1.IN.Aut AND "STATUS_2R1".RO01.Main.AutoRun AND "STATUS_2R2".RO01.Main.AutoRun AND NOT "2R1+RC01_In".SpdRdce AND NOT "2R2+RC01_In".SpdRdce AND ((("2R1+RC01_App_In".PosStanbyOUT OR "STATUS_2R1".NotUsed) AND "2R2+RC01_App_In".PosStanbyOUT) OR (("2R1+RC01_App_In".PosStanbyIN OR "STATUS_2R1".NotUsed) AND "2R2+RC01_App_In".PosStanbyIN)) AND "STATUS_Zone200".Mode.Specific.AutStart) OR ("JKComm_14" AND "STATUS_2R1"."000UH11-SF08"),   // TP
                  PT := #CT_StartPulse);
   "Communication".SCH1.OUT.StartPress := #ST_StartPulse.Q;
END_REGION

REGION Network 47: Immediately stop ram movement
   // FALSE = Immediately stop
   RUNG wire#powerrail
      I_Contact( "STATUS_2R1".RO01.Specific.CollDetect )
      wire#w1
      I_Contact( "STATUS_2R2".RO01.Specific.CollDetect )
      wire#w2
      I_Contact( "STATUS_2R1".RO01_LubStartErr.Main.CollErr )
      I_Contact( "STATUS_2R2".RO01_LubStartErr.Main.CollErr )
      I_Contact( "STATUS_Zone200"."RU01-QQ01".Specific.RequestPause )
      I_Contact( "STATUS_Zone200"."RU01-QQ02".Specific.RequestPause )
      I_Contact( "STATUS_Zone200"."RU01-QQ03".Specific.RequestPause )
      I_Contact( "STATUS_Zone200"."RU01-QQ04".Specific.RequestPause )
      I_Contact( "STATUS_Zone200"."RU01-QQ05".Specific.RequestPause )
      Contact( "STATUS_2R1"."000UH11-SF12" )
      Coil( "Communication".SCH1.OUT.IS )
   END_RUNG
   RUNG wire#powerrail
      Contact( "STATUS_2R1".RO01.Specific.ZoneRel.Zone[1].Rel )
   END_RUNG wire#w1
   RUNG wire#w1
      Contact( "STATUS_2R2".RO01.Specific.ZoneRel.Zone[1].Rel )
   END_RUNG wire#w2
   // the same network as SCL:
   "Communication".SCH1.OUT.IS := (NOT "STATUS_2R1".RO01.Specific.CollDetect OR "STATUS_2R1".RO01.Specific.ZoneRel.Zone[1].Rel) AND (NOT "STATUS_2R2".RO01.Specific.CollDetect OR "STATUS_2R2".RO01.Specific.ZoneRel.Zone[1].Rel) AND NOT "STATUS_2R1".RO01_LubStartErr.Main.CollErr AND NOT "STATUS_2R2".RO01_LubStartErr.Main.CollErr AND NOT "STATUS_Zone200"."RU01-QQ01".Specific.RequestPause AND NOT "STATUS_Zone200"."RU01-QQ02".Specific.RequestPause AND NOT "STATUS_Zone200"."RU01-QQ03".Specific.RequestPause AND NOT "STATUS_Zone200"."RU01-QQ04".Specific.RequestPause AND NOT "STATUS_Zone200"."RU01-QQ05".Specific.RequestPause AND "STATUS_2R1"."000UH11-SF12";
END_REGION

REGION Network 48: Control
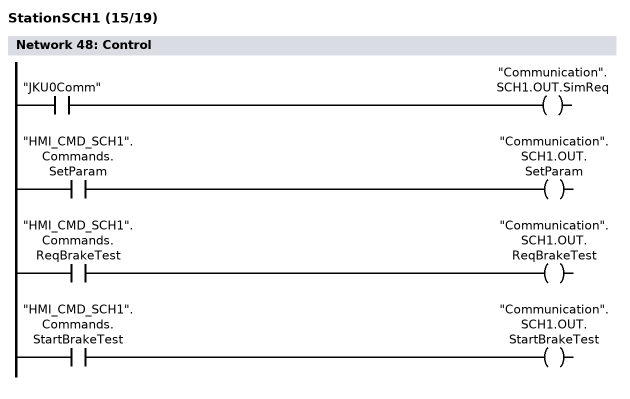
   RUNG wire#powerrail
      Contact( "JKU0Comm" )
      Coil( "Communication".SCH1.OUT.SimReq )
   END_RUNG
   RUNG wire#powerrail
      Contact( "HMI_CMD_SCH1".Commands.SetParam )
      Coil( "Communication".SCH1.OUT.SetParam )
   END_RUNG
   RUNG wire#powerrail
      Contact( "HMI_CMD_SCH1".Commands.ReqBrakeTest )
      Coil( "Communication".SCH1.OUT.ReqBrakeTest )
   END_RUNG
   RUNG wire#powerrail
      Contact( "HMI_CMD_SCH1".Commands.StartBrakeTest )
      Coil( "Communication".SCH1.OUT.StartBrakeTest )
   END_RUNG
   // the same network as SCL:
   "Communication".SCH1.OUT.SimReq := "JKU0Comm";
   "Communication".SCH1.OUT.SetParam := "HMI_CMD_SCH1".Commands.SetParam;
   "Communication".SCH1.OUT.ReqBrakeTest := "HMI_CMD_SCH1".Commands.ReqBrakeTest;
   "Communication".SCH1.OUT.StartBrakeTest := "HMI_CMD_SCH1".Commands.StartBrakeTest;
END_REGION

REGION Network 49: Lubrication
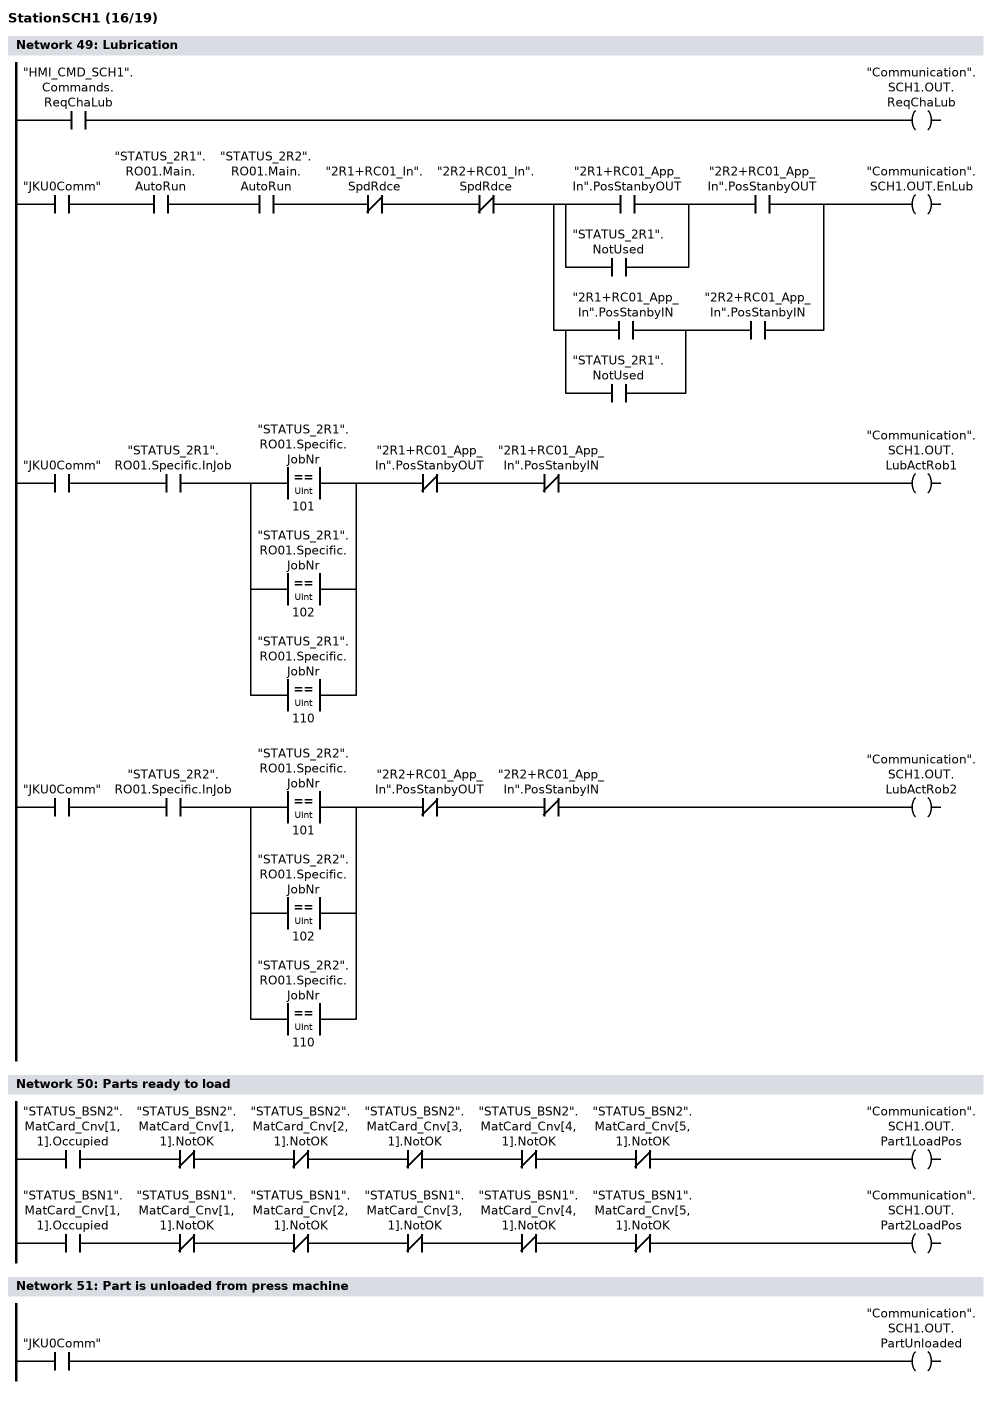
   RUNG wire#powerrail
      Contact( "HMI_CMD_SCH1".Commands.ReqChaLub )
      Coil( "Communication".SCH1.OUT.ReqChaLub )
   END_RUNG
   RUNG wire#powerrail
      Contact( "JKU0Comm" )
      Contact( "STATUS_2R1".RO01.Main.AutoRun )
      Contact( "STATUS_2R2".RO01.Main.AutoRun )
      I_Contact( "2R1+RC01_In".SpdRdce )
      I_Contact( "2R2+RC01_In".SpdRdce )
      wire#w1
      Contact( "2R1+RC01_App_In".PosStanbyOUT )
      wire#w2
      Contact( "2R2+RC01_App_In".PosStanbyOUT )
      wire#w3
      Coil( "Communication".SCH1.OUT.EnLub )
   END_RUNG
   RUNG wire#w1
      Contact( "STATUS_2R1".NotUsed )
   END_RUNG wire#w2
   RUNG wire#w1
      Contact( "2R1+RC01_App_In".PosStanbyIN )
      wire#w4
      Contact( "2R2+RC01_App_In".PosStanbyIN )
   END_RUNG wire#w3
   RUNG wire#w1
      Contact( "STATUS_2R1".NotUsed )
   END_RUNG wire#w4
   RUNG wire#powerrail
      Contact( "JKU0Comm" )
      Contact( "STATUS_2R1".RO01.Specific.InJob )
      wire#w5
      { S7_Templates := "SrcType := UInt" } EQ_Contact(in1 := "STATUS_2R1".RO01.Specific.JobNr, in2 := 101)
      wire#w6
      I_Contact( "2R1+RC01_App_In".PosStanbyOUT )
      I_Contact( "2R1+RC01_App_In".PosStanbyIN )
      Coil( "Communication".SCH1.OUT.LubActRob1 )
   END_RUNG
   RUNG wire#w5
      { S7_Templates := "SrcType := UInt" } EQ_Contact(in1 := "STATUS_2R1".RO01.Specific.JobNr, in2 := 102)
   END_RUNG wire#w6
   RUNG wire#w5
      { S7_Templates := "SrcType := UInt" } EQ_Contact(in1 := "STATUS_2R1".RO01.Specific.JobNr, in2 := 110)
   END_RUNG wire#w6
   RUNG wire#powerrail
      Contact( "JKU0Comm" )
      Contact( "STATUS_2R2".RO01.Specific.InJob )
      wire#w7
      { S7_Templates := "SrcType := UInt" } EQ_Contact(in1 := "STATUS_2R2".RO01.Specific.JobNr, in2 := 101)
      wire#w8
      I_Contact( "2R2+RC01_App_In".PosStanbyOUT )
      I_Contact( "2R2+RC01_App_In".PosStanbyIN )
      Coil( "Communication".SCH1.OUT.LubActRob2 )
   END_RUNG
   RUNG wire#w7
      { S7_Templates := "SrcType := UInt" } EQ_Contact(in1 := "STATUS_2R2".RO01.Specific.JobNr, in2 := 102)
   END_RUNG wire#w8
   RUNG wire#w7
      { S7_Templates := "SrcType := UInt" } EQ_Contact(in1 := "STATUS_2R2".RO01.Specific.JobNr, in2 := 110)
   END_RUNG wire#w8
   // the same network as SCL:
   "Communication".SCH1.OUT.ReqChaLub := "HMI_CMD_SCH1".Commands.ReqChaLub;
   "Communication".SCH1.OUT.EnLub := "JKU0Comm" AND "STATUS_2R1".RO01.Main.AutoRun AND "STATUS_2R2".RO01.Main.AutoRun AND NOT "2R1+RC01_In".SpdRdce AND NOT "2R2+RC01_In".SpdRdce AND ((("2R1+RC01_App_In".PosStanbyOUT OR "STATUS_2R1".NotUsed) AND "2R2+RC01_App_In".PosStanbyOUT) OR (("2R1+RC01_App_In".PosStanbyIN OR "STATUS_2R1".NotUsed) AND "2R2+RC01_App_In".PosStanbyIN));
   "Communication".SCH1.OUT.LubActRob1 := "JKU0Comm" AND "STATUS_2R1".RO01.Specific.InJob AND (("STATUS_2R1".RO01.Specific.JobNr = 101) OR ("STATUS_2R1".RO01.Specific.JobNr = 102) OR ("STATUS_2R1".RO01.Specific.JobNr = 110)) AND NOT "2R1+RC01_App_In".PosStanbyOUT AND NOT "2R1+RC01_App_In".PosStanbyIN;
   "Communication".SCH1.OUT.LubActRob2 := "JKU0Comm" AND "STATUS_2R2".RO01.Specific.InJob AND (("STATUS_2R2".RO01.Specific.JobNr = 101) OR ("STATUS_2R2".RO01.Specific.JobNr = 102) OR ("STATUS_2R2".RO01.Specific.JobNr = 110)) AND NOT "2R2+RC01_App_In".PosStanbyOUT AND NOT "2R2+RC01_App_In".PosStanbyIN;
END_REGION

REGION Network 50: Parts ready to load
   RUNG wire#powerrail
      Contact( "STATUS_BSN2".MatCard_Cnv[1, 1].Occupied )
      I_Contact( "STATUS_BSN2".MatCard_Cnv[1, 1].NotOK )
      I_Contact( "STATUS_BSN2".MatCard_Cnv[2, 1].NotOK )
      I_Contact( "STATUS_BSN2".MatCard_Cnv[3, 1].NotOK )
      I_Contact( "STATUS_BSN2".MatCard_Cnv[4, 1].NotOK )
      I_Contact( "STATUS_BSN2".MatCard_Cnv[5, 1].NotOK )
      Coil( "Communication".SCH1.OUT.Part1LoadPos )
   END_RUNG
   RUNG wire#powerrail
      Contact( "STATUS_BSN1".MatCard_Cnv[1, 1].Occupied )
      I_Contact( "STATUS_BSN1".MatCard_Cnv[1, 1].NotOK )
      I_Contact( "STATUS_BSN1".MatCard_Cnv[2, 1].NotOK )
      I_Contact( "STATUS_BSN1".MatCard_Cnv[3, 1].NotOK )
      I_Contact( "STATUS_BSN1".MatCard_Cnv[4, 1].NotOK )
      I_Contact( "STATUS_BSN1".MatCard_Cnv[5, 1].NotOK )
      Coil( "Communication".SCH1.OUT.Part2LoadPos )
   END_RUNG
   // the same network as SCL:
   "Communication".SCH1.OUT.Part1LoadPos := "STATUS_BSN2".MatCard_Cnv[1, 1].Occupied AND NOT "STATUS_BSN2".MatCard_Cnv[1, 1].NotOK AND NOT "STATUS_BSN2".MatCard_Cnv[2, 1].NotOK AND NOT "STATUS_BSN2".MatCard_Cnv[3, 1].NotOK AND NOT "STATUS_BSN2".MatCard_Cnv[4, 1].NotOK AND NOT "STATUS_BSN2".MatCard_Cnv[5, 1].NotOK;
   "Communication".SCH1.OUT.Part2LoadPos := "STATUS_BSN1".MatCard_Cnv[1, 1].Occupied AND NOT "STATUS_BSN1".MatCard_Cnv[1, 1].NotOK AND NOT "STATUS_BSN1".MatCard_Cnv[2, 1].NotOK AND NOT "STATUS_BSN1".MatCard_Cnv[3, 1].NotOK AND NOT "STATUS_BSN1".MatCard_Cnv[4, 1].NotOK AND NOT "STATUS_BSN1".MatCard_Cnv[5, 1].NotOK;
END_REGION

REGION Network 51: Part is unloaded from press machine
   RUNG wire#powerrail
      Contact( "JKU0Comm" )
      Coil( "Communication".SCH1.OUT.PartUnloaded )
   END_RUNG
   // the same network as SCL:
   "Communication".SCH1.OUT.PartUnloaded := "JKU0Comm";
END_REGION

REGION Network 52: Part to die request
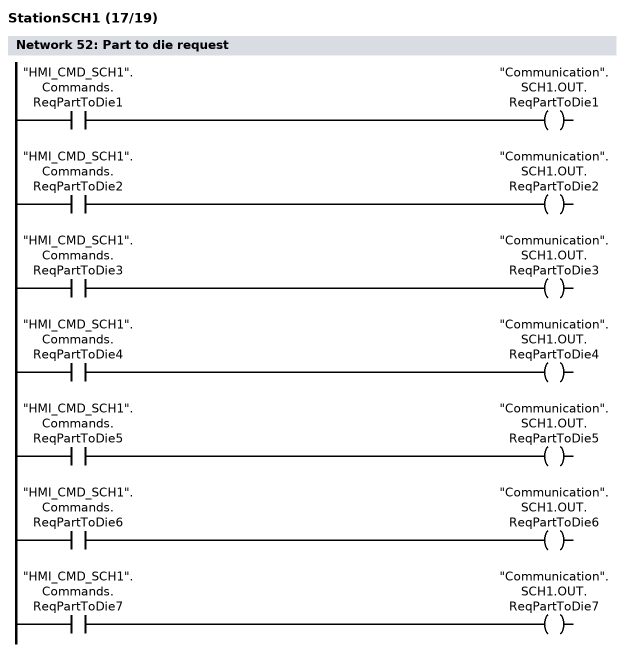
   RUNG wire#powerrail
      Contact( "HMI_CMD_SCH1".Commands.ReqPartToDie1 )
      Coil( "Communication".SCH1.OUT.ReqPartToDie1 )
   END_RUNG
   RUNG wire#powerrail
      Contact( "HMI_CMD_SCH1".Commands.ReqPartToDie2 )
      Coil( "Communication".SCH1.OUT.ReqPartToDie2 )
   END_RUNG
   RUNG wire#powerrail
      Contact( "HMI_CMD_SCH1".Commands.ReqPartToDie3 )
      Coil( "Communication".SCH1.OUT.ReqPartToDie3 )
   END_RUNG
   RUNG wire#powerrail
      Contact( "HMI_CMD_SCH1".Commands.ReqPartToDie4 )
      Coil( "Communication".SCH1.OUT.ReqPartToDie4 )
   END_RUNG
   RUNG wire#powerrail
      Contact( "HMI_CMD_SCH1".Commands.ReqPartToDie5 )
      Coil( "Communication".SCH1.OUT.ReqPartToDie5 )
   END_RUNG
   RUNG wire#powerrail
      Contact( "HMI_CMD_SCH1".Commands.ReqPartToDie6 )
      Coil( "Communication".SCH1.OUT.ReqPartToDie6 )
   END_RUNG
   RUNG wire#powerrail
      Contact( "HMI_CMD_SCH1".Commands.ReqPartToDie7 )
      Coil( "Communication".SCH1.OUT.ReqPartToDie7 )
   END_RUNG
   // the same network as SCL:
   "Communication".SCH1.OUT.ReqPartToDie1 := "HMI_CMD_SCH1".Commands.ReqPartToDie1;
   "Communication".SCH1.OUT.ReqPartToDie2 := "HMI_CMD_SCH1".Commands.ReqPartToDie2;
   "Communication".SCH1.OUT.ReqPartToDie3 := "HMI_CMD_SCH1".Commands.ReqPartToDie3;
   "Communication".SCH1.OUT.ReqPartToDie4 := "HMI_CMD_SCH1".Commands.ReqPartToDie4;
   "Communication".SCH1.OUT.ReqPartToDie5 := "HMI_CMD_SCH1".Commands.ReqPartToDie5;
   "Communication".SCH1.OUT.ReqPartToDie6 := "HMI_CMD_SCH1".Commands.ReqPartToDie6;
   "Communication".SCH1.OUT.ReqPartToDie7 := "HMI_CMD_SCH1".Commands.ReqPartToDie7;
END_REGION

REGION Network 53: Request for open stopper on press infeed
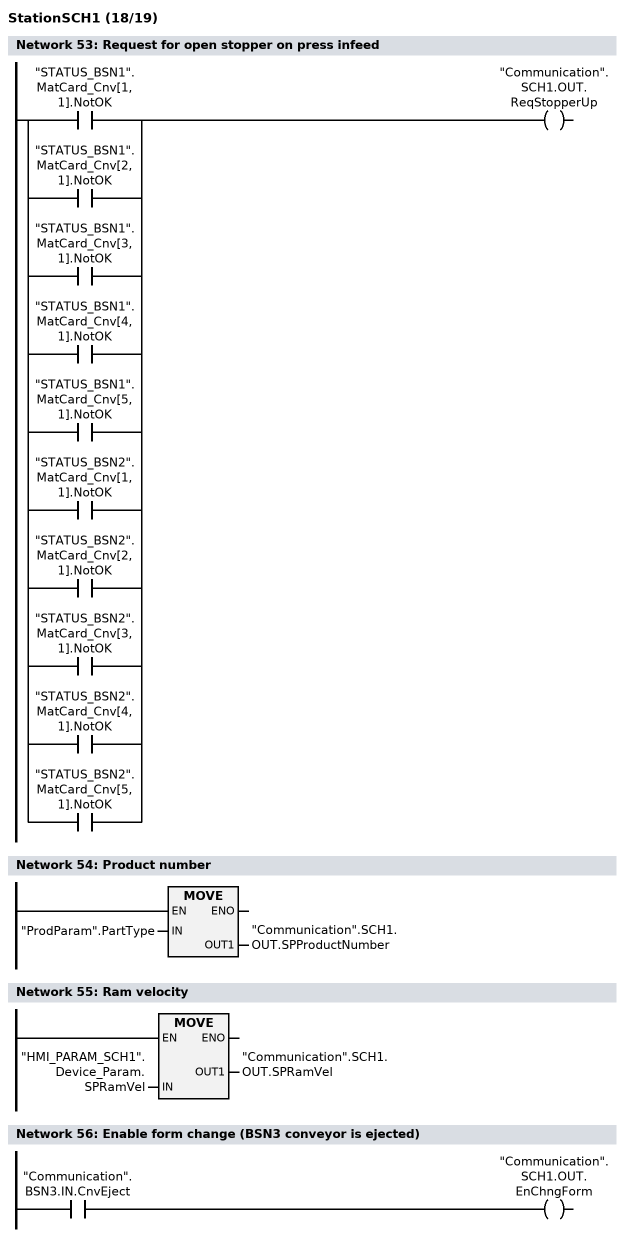
   RUNG wire#powerrail
      Contact( "STATUS_BSN1".MatCard_Cnv[1, 1].NotOK )
      wire#w1
      Coil( "Communication".SCH1.OUT.ReqStopperUp )
   END_RUNG
   RUNG wire#powerrail
      Contact( "STATUS_BSN1".MatCard_Cnv[2, 1].NotOK )
   END_RUNG wire#w1
   RUNG wire#powerrail
      Contact( "STATUS_BSN1".MatCard_Cnv[3, 1].NotOK )
   END_RUNG wire#w1
   RUNG wire#powerrail
      Contact( "STATUS_BSN1".MatCard_Cnv[4, 1].NotOK )
   END_RUNG wire#w1
   RUNG wire#powerrail
      Contact( "STATUS_BSN1".MatCard_Cnv[5, 1].NotOK )
   END_RUNG wire#w1
   RUNG wire#powerrail
      Contact( "STATUS_BSN2".MatCard_Cnv[1, 1].NotOK )
   END_RUNG wire#w1
   RUNG wire#powerrail
      Contact( "STATUS_BSN2".MatCard_Cnv[2, 1].NotOK )
   END_RUNG wire#w1
   RUNG wire#powerrail
      Contact( "STATUS_BSN2".MatCard_Cnv[3, 1].NotOK )
   END_RUNG wire#w1
   RUNG wire#powerrail
      Contact( "STATUS_BSN2".MatCard_Cnv[4, 1].NotOK )
   END_RUNG wire#w1
   RUNG wire#powerrail
      Contact( "STATUS_BSN2".MatCard_Cnv[5, 1].NotOK )
   END_RUNG wire#w1
   // the same network as SCL:
   "Communication".SCH1.OUT.ReqStopperUp := "STATUS_BSN1".MatCard_Cnv[1, 1].NotOK OR "STATUS_BSN1".MatCard_Cnv[2, 1].NotOK OR "STATUS_BSN1".MatCard_Cnv[3, 1].NotOK OR "STATUS_BSN1".MatCard_Cnv[4, 1].NotOK OR "STATUS_BSN1".MatCard_Cnv[5, 1].NotOK OR "STATUS_BSN2".MatCard_Cnv[1, 1].NotOK OR "STATUS_BSN2".MatCard_Cnv[2, 1].NotOK OR "STATUS_BSN2".MatCard_Cnv[3, 1].NotOK OR "STATUS_BSN2".MatCard_Cnv[4, 1].NotOK OR "STATUS_BSN2".MatCard_Cnv[5, 1].NotOK;
END_REGION

REGION Network 54: Product number
   RUNG wire#powerrail
      Move(in := "ProdParam".PartType, out1 => "Communication".SCH1.OUT.SPProductNumber)
   END_RUNG
   // the same network as SCL:
   "Communication".SCH1.OUT.SPProductNumber := "ProdParam".PartType;
END_REGION

REGION Network 55: Ram velocity
   RUNG wire#powerrail
      Move(in := "HMI_PARAM_SCH1".Device_Param.SPRamVel, out1 => "Communication".SCH1.OUT.SPRamVel)
   END_RUNG
   // the same network as SCL:
   "Communication".SCH1.OUT.SPRamVel := "HMI_PARAM_SCH1".Device_Param.SPRamVel;
END_REGION

REGION Network 56: Enable form change (BSN3 conveyor is ejected)
   RUNG wire#powerrail
      Contact( "Communication".BSN3.IN.CnvEject )
      Coil( "Communication".SCH1.OUT.EnChngForm )
   END_RUNG
   // the same network as SCL:
   "Communication".SCH1.OUT.EnChngForm := "Communication".BSN3.IN.CnvEject;
END_REGION

REGION Network 57: *************** Signalization ***************
END_REGION

REGION Network 58: HW switches - Press blocking
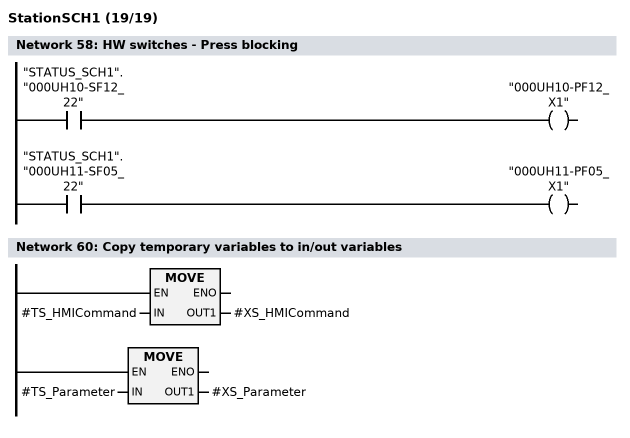
   RUNG wire#powerrail
      Contact( "STATUS_SCH1"."000UH10-SF12_22" )
      Coil( "000UH10-PF12_X1" )
   END_RUNG
   RUNG wire#powerrail
      Contact( "STATUS_SCH1"."000UH11-SF05_22" )
      Coil( "000UH11-PF05_X1" )
   END_RUNG
   // the same network as SCL:
   "000UH10-PF12_X1" := "STATUS_SCH1"."000UH10-SF12_22";
   "000UH11-PF05_X1" := "STATUS_SCH1"."000UH11-SF05_22";
END_REGION

REGION Network 59: *************** End ***************
END_REGION

REGION Network 60: Copy temporary variables to in/out variables
   RUNG wire#powerrail
      Move(in := #TS_HMICommand, out1 => #XS_HMICommand)
   END_RUNG
   RUNG wire#powerrail
      Move(in := #TS_Parameter, out1 => #XS_Parameter)
   END_RUNG
   // the same network as SCL:
   #XS_HMICommand := #TS_HMICommand;
   #XS_Parameter := #TS_Parameter;
END_REGION
END_FUNCTION_BLOCK
